LIN {X 0,Y 411.309,Z 303.251,A -85,B 0,C 180,E1 -10615.099,E2 -10615.099} C_VEL
LIN {X 0,Y 411.516,Z 303.227,A -85,B 0,C 180,E1 -10618.042,E2 -10618.042} C_VEL
LIN {X 0,Y 411.646,Z 303.212,A -85,B 0,C 180,E1 -10620,E2 -10620} C_VEL
LIN {X 0,Y 411.47,Z 303.233,A -85,B 0,C 180,E1 -10622.937,E2 -10622.937} C_VEL
LIN {X 0,Y 411.429,Z 303.238,A -85,B 0,C 180,E1 -10626.867,E2 -10626.867} C_VEL
LIN {X 0,Y 411.156,Z 303.275,A -85,B 0,C 180,E1 -10629.842,E2 -10629.842} C_VEL
LIN {X 0,Y 411.049,Z 303.289,A -85,B 0,C 180,E1 -10630.84,E2 -10630.84} C_VEL
LIN {X 0,Y 411.031,Z 303.714,A -85,B 0,C 180,E1 -10631.84,E2 -10631.84} C_VEL
LIN {X 0,Y 410.866,Z 306.355,A -85,B 0,C 180,E1 -10634.867,E2 -10634.867} C_VEL
LIN {X 0,Y 410.709,Z 309.078,A -85,B 0,C 180,E1 -10637.939,E2 -10637.939} C_VEL
LIN {X 0,Y 410.69,Z 311.358,A -85,B 0,C 180,E1 -10640.34,E2 -10640.34} C_VEL
LIN {X 0,Y 414.787,Z 325.038,A -85,B 0,C 180,E1 -10641.071,E2 -10641.071} C_VEL
LIN {X 0,Y 416.146,Z 330.89,A -85,B 0,C 180,E1 -10641.434,E2 -10641.434} C_VEL
LIN {X 0,Y 415.65,Z 342.021,A -85,B 0,C 180,E1 -10642.099,E2 -10642.099} C_VEL
LIN {X 0,Y 414.871,Z 354.086,A -85,B 0,C 180,E1 -10643.037,E2 -10643.037} C_VEL
LIN {X 0,Y 414.058,Z 365.557,A -85,B 0,C 180,E1 -10644.172,E2 -10644.172} C_VEL
LIN {X 0,Y 413.296,Z 375.312,A -85,B 0,C 180,E1 -10645.388,E2 -10645.388} C_VEL
LIN {X 0,Y 412.511,Z 384.696,A -85,B 0,C 180,E1 -10646.839,E2 -10646.839} C_VEL
LIN {X 0,Y 411.876,Z 392.147,A -85,B 0,C 180,E1 -10648.272,E2 -10648.272} C_VEL
LIN {X 0,Y 411.372,Z 398.098,A -85,B 0,C 180,E1 -10649.699,E2 -10649.699} C_VEL
LIN {X 0,Y 410.927,Z 403.134,A -85,B 0,C 180,E1 -10651.224,E2 -10651.224} C_VEL
LIN {X 0,Y 410.575,Z 407.484,A -85,B 0,C 180,E1 -10652.99,E2 -10652.99} C_VEL
LIN {X 0,Y 410.282,Z 410.333,A -85,B 0,C 180,E1 -10654.691,E2 -10654.691} C_VEL
LIN {X 0,Y 410.113,Z 411.91,A -85,B 0,C 180,E1 -10656.348,E2 -10656.348} C_VEL
LIN {X 0,Y 410.08,Z 412.317,A -85,B 0,C 180,E1 -10658.095,E2 -10658.095} C_VEL
LIN {X 0,Y 410.112,Z 411.728,A -85,B 0,C 180,E1 -10659.542,E2 -10659.542} C_VEL
LIN {X 0,Y 410.193,Z 410.148,A -85,B 0,C 180,E1 -10661.073,E2 -10661.073} C_VEL
LIN {X 0,Y 410.43,Z 407.6,A -85,B 0,C 180,E1 -10662.581,E2 -10662.581} C_VEL
LIN {X 0,Y 410.647,Z 404.145,A -85,B 0,C 180,E1 -10664.043,E2 -10664.043} C_VEL
LIN {X 0,Y 410.959,Z 399.707,A -85,B 0,C 180,E1 -10665.479,E2 -10665.479} C_VEL
LIN {X 0,Y 411.253,Z 394.299,A -85,B 0,C 180,E1 -10666.876,E2 -10666.876} C_VEL
LIN {X 0,Y 411.824,Z 386.807,A -85,B 0,C 180,E1 -10668.418,E2 -10668.418} C_VEL
LIN {X 0,Y 412.453,Z 377.956,A -85,B 0,C 180,E1 -10669.879,E2 -10669.879} C_VEL
LIN {X 0,Y 413.129,Z 368.681,A -85,B 0,C 180,E1 -10671.121,E2 -10671.121} C_VEL
LIN {X 0,Y 413.823,Z 358.621,A -85,B 0,C 180,E1 -10672.209,E2 -10672.209} C_VEL
LIN {X 0,Y 414.436,Z 347.453,A -85,B 0,C 180,E1 -10673.186,E2 -10673.186} C_VEL
LIN {X 0,Y 415.151,Z 335.294,A -85,B 0,C 180,E1 -10674.014,E2 -10674.014} C_VEL
LIN {X 0,Y 415.255,Z 328.945,A -85,B 0,C 180,E1 -10674.367,E2 -10674.367} C_VEL
LIN {X 0,Y 412.168,Z 315.956,A -85,B 0,C 180,E1 -10675.058,E2 -10675.058} C_VEL
LIN {X 0,Y 410.372,Z 308.871,A -85,B 0,C 180,E1 -10675.373,E2 -10675.373} C_VEL
LIN {X 0,Y 410.408,Z 305.017,A -85,B 0,C 180,E1 -10679.087,E2 -10679.087} C_VEL
LIN {X 0,Y 410.466,Z 303.359,A -85,B 0,C 180,E1 -10680.835,E2 -10680.835} C_VEL
LIN {X 0,Y 410.797,Z 303.317,A -85,B 0,C 180,E1 -10683.588,E2 -10683.588} C_VEL
LIN {X 0,Y 411.124,Z 303.275,A -85,B 0,C 180,E1 -10686.848,E2 -10686.848} C_VEL
LIN {X 0,Y 411.215,Z 303.26,A -85,B 0,C 180,E1 -10690.051,E2 -10690.051} C_VEL
LIN {X 0,Y 411.264,Z 303.258,A -85,B 0,C 180,E1 -10693.131,E2 -10693.131} C_VEL
LIN {X 0,Y 411.307,Z 303.253,A -85,B 0,C 180,E1 -10696.896,E2 -10696.896} C_VEL
LIN {X 0,Y 411.293,Z 303.252,A -85,B 0,C 180,E1 -10700.161,E2 -10700.161} C_VEL
LIN {X 0,Y 411.424,Z 303.238,A -85,B 0,C 180,E1 -10703.132,E2 -10703.132} C_VEL
LIN {X 0,Y 411.308,Z 303.253,A -85,B 0,C 180,E1 -10705.099,E2 -10705.099} C_VEL
LIN {X 0,Y 411.512,Z 303.225,A -85,B 0,C 180,E1 -10708.043,E2 -10708.043} C_VEL
LIN {X 0,Y 411.642,Z 303.208,A -85,B 0,C 180,E1 -10710,E2 -10710} C_VEL
LIN {X 0,Y 411.467,Z 303.234,A -85,B 0,C 180,E1 -10712.937,E2 -10712.937} C_VEL
LIN {X 0,Y 411.339,Z 303.246,A -85,B 0,C 180,E1 -10715.221,E2 -10715.221} C_VEL
LIN {X 0,Y 410.74,Z 303.323,A -85,B 0,C 180,E1 -10716.039,E2 -10716.039} C_VEL
LIN {X 0,Y 407.884,Z 303.676,A -85,B 0,C 180,E1 -10717.368,E2 -10717.368} C_VEL
LIN {X 0,Y 405.417,Z 303.987,A -85,B 0,C 180,E1 -10718.442,E2 -10718.442} C_VEL
LIN {X 0,Y 404.347,Z 304.117,A -85,B 0,C 180,E1 -10719.272,E2 -10719.272} C_VEL
LIN {X 0,Y 404.257,Z 304.128,A -85,B 0,C 180,E1 -10719.554,E2 -10719.554} C_VEL
LIN {X 0,Y 404.267,Z 304.127,A -85,B 0,C 180,E1 -10723.211,E2 -10723.211} C_VEL
LIN {X 0,Y 404.217,Z 304.134,A -85,B 0,C 180,E1 -10727.007,E2 -10727.007} C_VEL
LIN {X 0,Y 404.165,Z 304.143,A -85,B 0,C 180,E1 -10730.352,E2 -10730.352} C_VEL
LIN {X 0,Y 404.171,Z 304.139,A -85,B 0,C 180,E1 -10733.575,E2 -10733.575} C_VEL
LIN {X 0,Y 404.185,Z 304.139,A -85,B 0,C 180,E1 -10735.767,E2 -10735.767} C_VEL
LIN {X 0,Y 404.196,Z 304.139,A -85,B 0,C 180,E1 -10738,E2 -10738} C_VEL
LIN {X 0,Y 404.14,Z 304.144,A -85,B 0,C 180,E1 -10741.558,E2 -10741.558} C_VEL
LIN {X 0,Y 404.185,Z 304.137,A -85,B 0,C 180,E1 -10745.016,E2 -10745.016} C_VEL
LIN {X 0,Y 404.156,Z 304.141,A -85,B 0,C 180,E1 -10748.757,E2 -10748.757} C_VEL
LIN {X 0,Y 404.125,Z 304.148,A -85,B 0,C 180,E1 -10751.6,E2 -10751.6} C_VEL
LIN {X 0,Y 404.147,Z 304.142,A -85,B 0,C 180,E1 -10754.522,E2 -10754.522} C_VEL
LIN {X 0,Y 404.139,Z 304.144,A -85,B 0,C 180,E1 -10757.296,E2 -10757.296} C_VEL
LIN {X 0,Y 404.171,Z 304.142,A -85,B 0,C 180,E1 -10759.956,E2 -10759.956} C_VEL
LIN {X 0,Y 404.139,Z 304.144,A -85,B 0,C 180,E1 -10763.125,E2 -10763.125} C_VEL
LIN {X 0,Y 404.147,Z 304.142,A -85,B 0,C 180,E1 -10766.188,E2 -10766.188} C_VEL
LIN {X 0,Y 404.149,Z 304.144,A -85,B 0,C 180,E1 -10769.715,E2 -10769.715} C_VEL
LIN {X 0,Y 404.196,Z 304.138,A -85,B 0,C 180,E1 -10773.123,E2 -10773.123} C_VEL
LIN {X 0,Y 404.173,Z 304.142,A -85,B 0,C 180,E1 -10775.334,E2 -10775.334} C_VEL
LIN {X 0,Y 404.142,Z 304.142,A -85,B 0,C 180,E1 -10778.581,E2 -10778.581} C_VEL
LIN {X 0,Y 404.209,Z 304.135,A -85,B 0,C 180,E1 -10781.762,E2 -10781.762} C_VEL
LIN {X 0,Y 404.21,Z 304.136,A -85,B 0,C 180,E1 -10784.882,E2 -10784.882} C_VEL
LIN {X 0,Y 404.261,Z 304.128,A -85,B 0,C 180,E1 -10787.959,E2 -10787.959} C_VEL
LIN {X 0,Y 404.27,Z 304.13,A -85,B 0,C 180,E1 -10790.999,E2 -10790.999} C_VEL
LIN {X 0,Y 404.422,Z 304.107,A -85,B 0,C 180,E1 -10794.015,E2 -10794.015} C_VEL
LIN {X 0,Y 404.483,Z 304.099,A -85,B 0,C 180,E1 -10798.009,E2 -10798.009} C_VEL
LIN {X 0,Y 404.612,Z 304.084,A -85,B 0,C 180,E1 -10800,E2 -10800} C_VEL
LIN {X 0,Y 404.408,Z 304.112,A -85,B 0,C 180,E1 -10802.989,E2 -10802.989} C_VEL
LIN {X 0,Y 404.373,Z 304.116,A -85,B 0,C 180,E1 -10806.988,E2 -10806.988} C_VEL
LIN {X 0,Y 404.261,Z 304.127,A -85,B 0,C 180,E1 -10810.012,E2 -10810.012} C_VEL
LIN {X 0,Y 404.271,Z 304.126,A -85,B 0,C 180,E1 -10813.211,E2 -10813.211} C_VEL
LIN {X 0,Y 404.22,Z 304.133,A -85,B 0,C 180,E1 -10817.007,E2 -10817.007} C_VEL
LIN {X 0,Y 404.168,Z 304.142,A -85,B 0,C 180,E1 -10820.352,E2 -10820.352} C_VEL
LIN {X 0,Y 404.164,Z 304.14,A -85,B 0,C 180,E1 -10823.575,E2 -10823.575} C_VEL
LIN {X 0,Y 404.155,Z 304.142,A -85,B 0,C 180,E1 -10826.88,E2 -10826.88} C_VEL
LIN {X 0,Y 404.148,Z 304.145,A -85,B 0,C 180,E1 -10830.285,E2 -10830.285} C_VEL
LIN {X 0,Y 404.149,Z 304.143,A -85,B 0,C 180,E1 -10833.812,E2 -10833.812} C_VEL
LIN {X 0,Y 404.139,Z 304.142,A -85,B 0,C 180,E1 -10836.875,E2 -10836.875} C_VEL
LIN {X 0,Y 404.151,Z 304.144,A -85,B 0,C 180,E1 -10840.08,E2 -10840.08} C_VEL
LIN {X 0,Y 404.153,Z 304.144,A -85,B 0,C 180,E1 -10843.083,E2 -10843.083} C_VEL
LIN {X 0,Y 404.15,Z 304.142,A -85,B 0,C 180,E1 -10845.926,E2 -10845.926} C_VEL
LIN {X 0,Y 404.171,Z 304.244,A -85,B 0,C 180,E1 -10847.204,E2 -10847.204} C_VEL
LIN {X 0,Y 405.52,Z 311.584,A -85,B 0,C 180,E1 -10850.707,E2 -10850.707} C_VEL
LIN {X 0,Y 406.463,Z 317.496,A -85,B 0,C 180,E1 -10853.378,E2 -10853.378} C_VEL
LIN {X 0,Y 406.168,Z 323.082,A -85,B 0,C 180,E1 -10855.736,E2 -10855.736} C_VEL
LIN {X 0,Y 405.489,Z 330.3,A -85,B 0,C 180,E1 -10858.67,E2 -10858.67} C_VEL
LIN {X 0,Y 404.96,Z 337.41,A -85,B 0,C 180,E1 -10861.493,E2 -10861.493} C_VEL
LIN {X 0,Y 404.381,Z 345.551,A -85,B 0,C 180,E1 -10864.655,E2 -10864.655} C_VEL
LIN {X 0,Y 403.858,Z 354.455,A -85,B 0,C 180,E1 -10868.028,E2 -10868.028} C_VEL
LIN {X 0,Y 403.524,Z 362.939,A -85,B 0,C 180,E1 -10871.203,E2 -10871.203} C_VEL
LIN {X 0,Y 403.416,Z 365.913,A -85,B 0,C 180,E1 -10872.304,E2 -10872.304} C_VEL
LIN {X 0,Y 405.324,Z 379.721,A -85,B 0,C 180,E1 -10872.813,E2 -10872.813} C_VEL
LIN {X 0,Y 406.616,Z 391.696,A -85,B 0,C 180,E1 -10873.425,E2 -10873.425} C_VEL
LIN {X 0,Y 407.147,Z 400.281,A -85,B 0,C 180,E1 -10873.967,E2 -10873.967} C_VEL
LIN {X 0,Y 406.322,Z 411.995,A -85,B 0,C 180,E1 -10874.834,E2 -10874.834} C_VEL
LIN {X 0,Y 405.435,Z 423.753,A -85,B 0,C 180,E1 -10875.955,E2 -10875.955} C_VEL
LIN {X 0,Y 404.729,Z 434.257,A -85,B 0,C 180,E1 -10877.209,E2 -10877.209} C_VEL
LIN {X 0,Y 404.15,Z 442.777,A -85,B 0,C 180,E1 -10878.464,E2 -10878.464} C_VEL
LIN {X 0,Y 403.562,Z 451.09,A -85,B 0,C 180,E1 -10879.971,E2 -10879.971} C_VEL
LIN {X 0,Y 403.285,Z 457.801,A -85,B 0,C 180,E1 -10881.481,E2 -10881.481} C_VEL
LIN {X 0,Y 403.077,Z 463.139,A -85,B 0,C 180,E1 -10882.989,E2 -10882.989} C_VEL
LIN {X 0,Y 403.034,Z 467.281,A -85,B 0,C 180,E1 -10884.496,E2 -10884.496} C_VEL
LIN {X 0,Y 402.964,Z 470.331,A -85,B 0,C 180,E1 -10886,E2 -10886} C_VEL
LIN {X 0,Y 403.09,Z 471.836,A -85,B 0,C 180,E1 -10887.002,E2 -10887.002} C_VEL
LIN {X 0,Y 403.089,Z 472.867,A -85,B 0,C 180,E1 -10888.002,E2 -10888.002} C_VEL
LIN {X 0,Y 403.098,Z 473.495,A -85,B 0,C 180,E1 -10889.001,E2 -10889.001} C_VEL
LIN {X 0,Y 403.069,Z 473.721,A -85,B 0,C 180,E1 -10890,E2 -10890} C_VEL
LIN {X 0,Y 403.097,Z 473.538,A -85,B 0,C 180,E1 -10890.999,E2 -10890.999} C_VEL
LIN {X 0,Y 403.098,Z 471.88,A -85,B 0,C 180,E1 -10892.998,E2 -10892.998} C_VEL
LIN {X 0,Y 402.965,Z 470.435,A -85,B 0,C 180,E1 -10894,E2 -10894} C_VEL
LIN {X 0,Y 402.993,Z 467.431,A -85,B 0,C 180,E1 -10895.504,E2 -10895.504} C_VEL
LIN {X 0,Y 403.076,Z 463.375,A -85,B 0,C 180,E1 -10897.011,E2 -10897.011} C_VEL
LIN {X 0,Y 403.302,Z 457.185,A -85,B 0,C 180,E1 -10898.771,E2 -10898.771} C_VEL
LIN {X 0,Y 403.651,Z 450.416,A -85,B 0,C 180,E1 -10900.28,E2 -10900.28} C_VEL
LIN {X 0,Y 404.289,Z 442.056,A -85,B 0,C 180,E1 -10901.786,E2 -10901.786} C_VEL
LIN {X 0,Y 404.923,Z 433.557,A -85,B 0,C 180,E1 -10903.04,E2 -10903.04} C_VEL
LIN {X 0,Y 405.684,Z 423.173,A -85,B 0,C 180,E1 -10904.292,E2 -10904.292} C_VEL
LIN {X 0,Y 406.678,Z 411.581,A -85,B 0,C 180,E1 -10905.409,E2 -10905.409} C_VEL
LIN {X 0,Y 407.546,Z 400.302,A -85,B 0,C 180,E1 -10906.274,E2 -10906.274} C_VEL
LIN {X 0,Y 406.791,Z 387.739,A -85,B 0,C 180,E1 -10907.08,E2 -10907.08} C_VEL
LIN {X 0,Y 405.258,Z 374.108,A -85,B 0,C 180,E1 -10907.764,E2 -10907.764} C_VEL
LIN {X 0,Y 403.409,Z 363.522,A -85,B 0,C 180,E1 -10908.21,E2 -10908.21} C_VEL
LIN {X 0,Y 403.741,Z 354.769,A -85,B 0,C 180,E1 -10911.442,E2 -10911.442} C_VEL
LIN {X 0,Y 404.156,Z 346.259,A -85,B 0,C 180,E1 -10914.667,E2 -10914.667} C_VEL
LIN {X 0,Y 404.826,Z 336.442,A -85,B 0,C 180,E1 -10918.517,E2 -10918.517} C_VEL
LIN {X 0,Y 405.705,Z 326.904,A -85,B 0,C 180,E1 -10922.481,E2 -10922.481} C_VEL
LIN {X 0,Y 406.508,Z 318.939,A -85,B 0,C 180,E1 -10926.003,E2 -10926.003} C_VEL
LIN {X 0,Y 406.15,Z 315.059,A -85,B 0,C 180,E1 -10927.9,E2 -10927.9} C_VEL
LIN {X 0,Y 405.06,Z 308.803,A -85,B 0,C 180,E1 -10931.248,E2 -10931.248} C_VEL
LIN {X 0,Y 404.152,Z 304.149,A -85,B 0,C 180,E1 -10934.074,E2 -10934.074} C_VEL
LIN {X 0,Y 404.14,Z 304.151,A -85,B 0,C 180,E1 -10937.296,E2 -10937.296} C_VEL
LIN {X 0,Y 404.172,Z 304.144,A -85,B 0,C 180,E1 -10939.955,E2 -10939.955} C_VEL
LIN {X 0,Y 404.14,Z 304.145,A -85,B 0,C 180,E1 -10943.125,E2 -10943.125} C_VEL
LIN {X 0,Y 404.149,Z 304.145,A -85,B 0,C 180,E1 -10946.188,E2 -10946.188} C_VEL
LIN {X 0,Y 404.15,Z 304.144,A -85,B 0,C 180,E1 -10949.715,E2 -10949.715} C_VEL
LIN {X 0,Y 404.2,Z 304.138,A -85,B 0,C 180,E1 -10953.123,E2 -10953.123} C_VEL
LIN {X 0,Y 404.182,Z 304.137,A -85,B 0,C 180,E1 -10955.334,E2 -10955.334} C_VEL
LIN {X 0,Y 404.144,Z 304.145,A -85,B 0,C 180,E1 -10958.581,E2 -10958.581} C_VEL
LIN {X 0,Y 404.213,Z 304.135,A -85,B 0,C 180,E1 -10961.762,E2 -10961.762} C_VEL
LIN {X 0,Y 404.211,Z 304.134,A -85,B 0,C 180,E1 -10964.882,E2 -10964.882} C_VEL
LIN {X 0,Y 404.261,Z 304.131,A -85,B 0,C 180,E1 -10967.958,E2 -10967.958} C_VEL
LIN {X 0,Y 404.271,Z 304.128,A -85,B 0,C 180,E1 -10970.998,E2 -10970.998} C_VEL
LIN {X 0,Y 404.396,Z 304.113,A -85,B 0,C 180,E1 -10974.015,E2 -10974.015} C_VEL
LIN {X 0,Y 404.485,Z 304.103,A -85,B 0,C 180,E1 -10978.008,E2 -10978.008} C_VEL
LIN {X 0,Y 404.615,Z 304.088,A -85,B 0,C 180,E1 -10980,E2 -10980} C_VEL
LIN {X 0,Y 404.427,Z 304.111,A -85,B 0,C 180,E1 -10982.988,E2 -10982.988} C_VEL
LIN {X 0,Y 404.374,Z 304.117,A -85,B 0,C 180,E1 -10986.988,E2 -10986.988} C_VEL
LIN {X 0,Y 404.082,Z 304.156,A -85,B 0,C 180,E1 -10990.016,E2 -10990.016} C_VEL
LIN {X 0,Y 403.981,Z 304.169,A -85,B 0,C 180,E1 -10991.032,E2 -10991.032} C_VEL
LIN {X 0,Y 403.933,Z 305.806,A -85,B 0,C 180,E1 -10993.073,E2 -10993.073} C_VEL
LIN {X 0,Y 403.805,Z 308.477,A -85,B 0,C 180,E1 -10996.169,E2 -10996.169} C_VEL
LIN {X 0,Y 403.644,Z 311.846,A -85,B 0,C 180,E1 -10999.972,E2 -10999.972} C_VEL
LIN {X 0,Y 407.768,Z 325.499,A -85,B 0,C 180,E1 -11000.724,E2 -11000.724} C_VEL
LIN {X 0,Y 409.449,Z 332.857,A -85,B 0,C 180,E1 -11001.194,E2 -11001.194} C_VEL
LIN {X 0,Y 408.798,Z 344.75,A -85,B 0,C 180,E1 -11001.949,E2 -11001.949} C_VEL
LIN {X 0,Y 407.961,Z 356.799,A -85,B 0,C 180,E1 -11002.94,E2 -11002.94} C_VEL
LIN {X 0,Y 407.096,Z 367.899,A -85,B 0,C 180,E1 -11004.111,E2 -11004.111} C_VEL
LIN {X 0,Y 406.301,Z 377.329,A -85,B 0,C 180,E1 -11005.348,E2 -11005.348} C_VEL
LIN {X 0,Y 405.511,Z 386.203,A -85,B 0,C 180,E1 -11006.783,E2 -11006.783} C_VEL
LIN {X 0,Y 404.858,Z 393.389,A -85,B 0,C 180,E1 -11008.232,E2 -11008.232} C_VEL
LIN {X 0,Y 404.244,Z 400.049,A -85,B 0,C 180,E1 -11009.922,E2 -11009.922} C_VEL
LIN {X 0,Y 403.812,Z 404.806,A -85,B 0,C 180,E1 -11011.481,E2 -11011.481} C_VEL
LIN {X 0,Y 403.457,Z 408.806,A -85,B 0,C 180,E1 -11013.265,E2 -11013.265} C_VEL
LIN {X 0,Y 403.152,Z 411.47,A -85,B 0,C 180,E1 -11015.119,E2 -11015.119} C_VEL
LIN {X 0,Y 403.038,Z 412.625,A -85,B 0,C 180,E1 -11016.666,E2 -11016.666} C_VEL
LIN {X 0,Y 403.001,Z 412.81,A -85,B 0,C 180,E1 -11018.301,E2 -11018.301} C_VEL
LIN {X 0,Y 403.059,Z 411.724,A -85,B 0,C 180,E1 -11020.177,E2 -11020.177} C_VEL
LIN {X 0,Y 403.264,Z 409.029,A -85,B 0,C 180,E1 -11022.142,E2 -11022.142} C_VEL
LIN {X 0,Y 403.522,Z 406.175,A -85,B 0,C 180,E1 -11023.518,E2 -11023.518} C_VEL
LIN {X 0,Y 403.771,Z 402.298,A -85,B 0,C 180,E1 -11024.941,E2 -11024.941} C_VEL
LIN {X 0,Y 404.115,Z 396.265,A -85,B 0,C 180,E1 -11026.641,E2 -11026.641} C_VEL
LIN {X 0,Y 404.707,Z 388.687,A -85,B 0,C 180,E1 -11028.307,E2 -11028.307} C_VEL
LIN {X 0,Y 405.314,Z 380.596,A -85,B 0,C 180,E1 -11029.724,E2 -11029.724} C_VEL
LIN {X 0,Y 406.092,Z 370.467,A -85,B 0,C 180,E1 -11031.15,E2 -11031.15} C_VEL
LIN {X 0,Y 406.787,Z 360.994,A -85,B 0,C 180,E1 -11032.231,E2 -11032.231} C_VEL
LIN {X 0,Y 407.493,Z 349.174,A -85,B 0,C 180,E1 -11033.314,E2 -11033.314} C_VEL
LIN {X 0,Y 408.246,Z 337.049,A -85,B 0,C 180,E1 -11034.174,E2 -11034.174} C_VEL
LIN {X 0,Y 408.438,Z 330.329,A -85,B 0,C 180,E1 -11034.567,E2 -11034.567} C_VEL
LIN {X 0,Y 405.471,Z 317.829,A -85,B 0,C 180,E1 -11035.262,E2 -11035.262} C_VEL
LIN {X 0,Y 403.314,Z 309.34,A -85,B 0,C 180,E1 -11035.656,E2 -11035.656} C_VEL
LIN {X 0,Y 403.318,Z 306.271,A -85,B 0,C 180,E1 -11038.633,E2 -11038.633} C_VEL
LIN {X 0,Y 403.42,Z 304.237,A -85,B 0,C 180,E1 -11040.804,E2 -11040.804} C_VEL
LIN {X 0,Y 403.718,Z 304.199,A -85,B 0,C 180,E1 -11043.088,E2 -11043.088} C_VEL
LIN {X 0,Y 403.948,Z 304.171,A -85,B 0,C 180,E1 -11045.319,E2 -11045.319} C_VEL
LIN {X 0,Y 404.145,Z 304.144,A -85,B 0,C 180,E1 -11047.506,E2 -11047.506} C_VEL
LIN {X 0,Y 404.163,Z 304.141,A -85,B 0,C 180,E1 -11050.707,E2 -11050.707} C_VEL
LIN {X 0,Y 404.222,Z 304.132,A -85,B 0,C 180,E1 -11053.848,E2 -11053.848} C_VEL
LIN {X 0,Y 404.284,Z 304.128,A -85,B 0,C 180,E1 -11056.939,E2 -11056.939} C_VEL
LIN {X 0,Y 404.259,Z 304.128,A -85,B 0,C 180,E1 -11059.988,E2 -11059.988} C_VEL
LIN {X 0,Y 404.37,Z 304.117,A -85,B 0,C 180,E1 -11063.012,E2 -11063.012} C_VEL
LIN {X 0,Y 404.278,Z 304.129,A -85,B 0,C 180,E1 -11065.013,E2 -11065.013} C_VEL
LIN {X 0,Y 404.481,Z 304.101,A -85,B 0,C 180,E1 -11068.008,E2 -11068.008} C_VEL
LIN {X 0,Y 404.611,Z 304.084,A -85,B 0,C 180,E1 -11070,E2 -11070} C_VEL
LIN {X 0,Y 404.424,Z 304.11,A -85,B 0,C 180,E1 -11072.988,E2 -11072.988} C_VEL
LIN {X 0,Y 404.37,Z 304.116,A -85,B 0,C 180,E1 -11076.988,E2 -11076.988} C_VEL
LIN {X 0,Y 404.257,Z 304.128,A -85,B 0,C 180,E1 -11079.554,E2 -11079.554} C_VEL
LIN {X 0,Y 403.584,Z 304.215,A -85,B 0,C 180,E1 -11080.385,E2 -11080.385} C_VEL
LIN {X 0,Y 400.732,Z 304.567,A -85,B 0,C 180,E1 -11081.737,E2 -11081.737} C_VEL
LIN {X 0,Y 398.316,Z 304.87,A -85,B 0,C 180,E1 -11082.829,E2 -11082.829} C_VEL
LIN {X 0,Y 397.271,Z 304.998,A -85,B 0,C 180,E1 -11083.674,E2 -11083.674} C_VEL
LIN {X 0,Y 397.181,Z 305.009,A -85,B 0,C 180,E1 -11083.96,E2 -11083.96} C_VEL
LIN {X 0,Y 397.175,Z 305.01,A -85,B 0,C 180,E1 -11087.507,E2 -11087.507} C_VEL
LIN {X 0,Y 397.104,Z 305.021,A -85,B 0,C 180,E1 -11090.73,E2 -11090.73} C_VEL
LIN {X 0,Y 397.135,Z 305.018,A -85,B 0,C 180,E1 -11094.018,E2 -11094.018} C_VEL
LIN {X 0,Y 397.196,Z 305.007,A -85,B 0,C 180,E1 -11097.39,E2 -11097.39} C_VEL
LIN {X 0,Y 397.079,Z 305.022,A -85,B 0,C 180,E1 -11100.883,E2 -11100.883} C_VEL
LIN {X 0,Y 397.126,Z 305.018,A -85,B 0,C 180,E1 -11104.494,E2 -11104.494} C_VEL
LIN {X 0,Y 397.104,Z 305.022,A -85,B 0,C 180,E1 -11108.275,E2 -11108.275} C_VEL
LIN {X 0,Y 397.09,Z 305.02,A -85,B 0,C 180,E1 -11110.909,E2 -11110.909} C_VEL
LIN {X 0,Y 397.103,Z 305.022,A -85,B 0,C 180,E1 -11113.649,E2 -11113.649} C_VEL
LIN {X 0,Y 397.104,Z 305.019,A -85,B 0,C 180,E1 -11116.521,E2 -11116.521} C_VEL
LIN {X 0,Y 397.117,Z 305.018,A -85,B 0,C 180,E1 -11120.423,E2 -11120.423} C_VEL
LIN {X 0,Y 397.11,Z 305.019,A -85,B 0,C 180,E1 -11124.266,E2 -11124.266} C_VEL
LIN {X 0,Y 397.117,Z 305.017,A -85,B 0,C 180,E1 -11126.727,E2 -11126.727} C_VEL
LIN {X 0,Y 397.127,Z 305.016,A -85,B 0,C 180,E1 -11130.296,E2 -11130.296} C_VEL
LIN {X 0,Y 397.197,Z 305.007,A -85,B 0,C 180,E1 -11132.61,E2 -11132.61} C_VEL
LIN {X 0,Y 397.129,Z 305.017,A -85,B 0,C 180,E1 -11135.982,E2 -11135.982} C_VEL
LIN {X 0,Y 397.142,Z 305.017,A -85,B 0,C 180,E1 -11139.705,E2 -11139.705} C_VEL
LIN {X 0,Y 397.186,Z 305.011,A -85,B 0,C 180,E1 -11142.845,E2 -11142.845} C_VEL
LIN {X 0,Y 397.233,Z 305.004,A -85,B 0,C 180,E1 -11146.703,E2 -11146.703} C_VEL
LIN {X 0,Y 397.221,Z 305.004,A -85,B 0,C 180,E1 -11149.809,E2 -11149.809} C_VEL
LIN {X 0,Y 397.342,Z 304.992,A -85,B 0,C 180,E1 -11152.888,E2 -11152.888} C_VEL
LIN {X 0,Y 397.256,Z 305.004,A -85,B 0,C 180,E1 -11154.925,E2 -11154.925} C_VEL
LIN {X 0,Y 397.452,Z 304.975,A -85,B 0,C 180,E1 -11157.973,E2 -11157.973} C_VEL
LIN {X 0,Y 397.581,Z 304.96,A -85,B 0,C 180,E1 -11160,E2 -11160} C_VEL
LIN {X 0,Y 397.342,Z 304.992,A -85,B 0,C 180,E1 -11163.042,E2 -11163.042} C_VEL
LIN {X 0,Y 397.348,Z 304.988,A -85,B 0,C 180,E1 -11166.092,E2 -11166.092} C_VEL
LIN {X 0,Y 397.24,Z 305.003,A -85,B 0,C 180,E1 -11169.162,E2 -11169.162} C_VEL
LIN {X 0,Y 397.224,Z 305.007,A -85,B 0,C 180,E1 -11172.258,E2 -11172.258} C_VEL
LIN {X 0,Y 397.183,Z 305.009,A -85,B 0,C 180,E1 -11175.392,E2 -11175.392} C_VEL
LIN {X 0,Y 397.162,Z 305.015,A -85,B 0,C 180,E1 -11178.574,E2 -11178.574} C_VEL
LIN {X 0,Y 397.1,Z 305.019,A -85,B 0,C 180,E1 -11181.818,E2 -11181.818} C_VEL
LIN {X 0,Y 397.127,Z 305.015,A -85,B 0,C 180,E1 -11185.134,E2 -11185.134} C_VEL
LIN {X 0,Y 397.103,Z 305.022,A -85,B 0,C 180,E1 -11188.545,E2 -11188.545} C_VEL
LIN {X 0,Y 397.082,Z 305.025,A -85,B 0,C 180,E1 -11192.071,E2 -11192.071} C_VEL
LIN {X 0,Y 397.123,Z 305.018,A -85,B 0,C 180,E1 -11195.503,E2 -11195.503} C_VEL
LIN {X 0,Y 397.128,Z 305.016,A -85,B 0,C 180,E1 -11198.86,E2 -11198.86} C_VEL
LIN {X 0,Y 397.068,Z 305.026,A -85,B 0,C 180,E1 -11202.268,E2 -11202.268} C_VEL
LIN {X 0,Y 397.09,Z 305.021,A -85,B 0,C 180,E1 -11205.069,E2 -11205.069} C_VEL
LIN {X 0,Y 397.135,Z 305.125,A -85,B 0,C 180,E1 -11206.915,E2 -11206.915} C_VEL
LIN {X 0,Y 398.297,Z 311.423,A -85,B 0,C 180,E1 -11209.997,E2 -11209.997} C_VEL
LIN {X 0,Y 399.203,Z 316.543,A -85,B 0,C 180,E1 -11212.395,E2 -11212.395} C_VEL
LIN {X 0,Y 399.474,Z 320.201,A -85,B 0,C 180,E1 -11214.027,E2 -11214.027} C_VEL
LIN {X 0,Y 398.797,Z 328.225,A -85,B 0,C 180,E1 -11217.401,E2 -11217.401} C_VEL
LIN {X 0,Y 398.011,Z 336.929,A -85,B 0,C 180,E1 -11220.949,E2 -11220.949} C_VEL
LIN {X 0,Y 397.341,Z 345.686,A -85,B 0,C 180,E1 -11224.432,E2 -11224.432} C_VEL
LIN {X 0,Y 396.836,Z 353.898,A -85,B 0,C 180,E1 -11227.619,E2 -11227.619} C_VEL
LIN {X 0,Y 396.402,Z 363.804,A -85,B 0,C 180,E1 -11231.39,E2 -11231.39} C_VEL
LIN {X 0,Y 396.335,Z 365.45,A -85,B 0,C 180,E1 -11232.014,E2 -11232.014} C_VEL
LIN {X 0,Y 398.363,Z 379.828,A -85,B 0,C 180,E1 -11232.565,E2 -11232.565} C_VEL
LIN {X 0,Y 399.717,Z 393.011,A -85,B 0,C 180,E1 -11233.275,E2 -11233.275} C_VEL
LIN {X 0,Y 400.163,Z 401.143,A -85,B 0,C 180,E1 -11233.811,E2 -11233.811} C_VEL
LIN {X 0,Y 399.315,Z 412.488,A -85,B 0,C 180,E1 -11234.692,E2 -11234.692} C_VEL
LIN {X 0,Y 398.386,Z 424.219,A -85,B 0,C 180,E1 -11235.849,E2 -11235.849} C_VEL
LIN {X 0,Y 397.779,Z 433.458,A -85,B 0,C 180,E1 -11236.981,E2 -11236.981} C_VEL
LIN {X 0,Y 397.147,Z 442.037,A -85,B 0,C 180,E1 -11238.258,E2 -11238.258} C_VEL
LIN {X 0,Y 396.499,Z 450.384,A -85,B 0,C 180,E1 -11239.79,E2 -11239.79} C_VEL
LIN {X 0,Y 396.205,Z 457.127,A -85,B 0,C 180,E1 -11241.328,E2 -11241.328} C_VEL
LIN {X 0,Y 396.005,Z 462.496,A -85,B 0,C 180,E1 -11242.864,E2 -11242.864} C_VEL
LIN {X 0,Y 395.949,Z 466.665,A -85,B 0,C 180,E1 -11244.398,E2 -11244.398} C_VEL
LIN {X 0,Y 395.882,Z 469.739,A -85,B 0,C 180,E1 -11245.928,E2 -11245.928} C_VEL
LIN {X 0,Y 396.002,Z 471.26,A -85,B 0,C 180,E1 -11246.948,E2 -11246.948} C_VEL
LIN {X 0,Y 396.015,Z 472.305,A -85,B 0,C 180,E1 -11247.966,E2 -11247.966} C_VEL
LIN {X 0,Y 396.046,Z 472.944,A -85,B 0,C 180,E1 -11248.983,E2 -11248.983} C_VEL
LIN {X 0,Y 396.016,Z 473.178,A -85,B 0,C 180,E1 -11250,E2 -11250} C_VEL
LIN {X 0,Y 396.028,Z 473.007,A -85,B 0,C 180,E1 -11251.017,E2 -11251.017} C_VEL
LIN {X 0,Y 395.998,Z 472.387,A -85,B 0,C 180,E1 -11252.034,E2 -11252.034} C_VEL
LIN {X 0,Y 396.01,Z 471.366,A -85,B 0,C 180,E1 -11253.052,E2 -11253.052} C_VEL
LIN {X 0,Y 395.883,Z 469.925,A -85,B 0,C 180,E1 -11254.072,E2 -11254.072} C_VEL
LIN {X 0,Y 395.894,Z 466.933,A -85,B 0,C 180,E1 -11255.603,E2 -11255.603} C_VEL
LIN {X 0,Y 396.004,Z 462.892,A -85,B 0,C 180,E1 -11257.136,E2 -11257.136} C_VEL
LIN {X 0,Y 396.22,Z 456.723,A -85,B 0,C 180,E1 -11258.929,E2 -11258.929} C_VEL
LIN {X 0,Y 396.601,Z 449.97,A -85,B 0,C 180,E1 -11260.465,E2 -11260.465} C_VEL
LIN {X 0,Y 397.314,Z 441.644,A -85,B 0,C 180,E1 -11261.996,E2 -11261.996} C_VEL
LIN {X 0,Y 398.098,Z 432.082,A -85,B 0,C 180,E1 -11263.425,E2 -11263.425} C_VEL
LIN {X 0,Y 398.861,Z 421.734,A -85,B 0,C 180,E1 -11264.672,E2 -11264.672} C_VEL
LIN {X 0,Y 399.964,Z 409.986,A -85,B 0,C 180,E1 -11265.805,E2 -11265.805} C_VEL
LIN {X 0,Y 400.669,Z 400.225,A -85,B 0,C 180,E1 -11266.561,E2 -11266.561} C_VEL
LIN {X 0,Y 399.967,Z 387.905,A -85,B 0,C 180,E1 -11267.381,E2 -11267.381} C_VEL
LIN {X 0,Y 398.35,Z 374.086,A -85,B 0,C 180,E1 -11268.103,E2 -11268.103} C_VEL
LIN {X 0,Y 396.351,Z 362.938,A -85,B 0,C 180,E1 -11268.583,E2 -11268.583} C_VEL
LIN {X 0,Y 396.715,Z 354.333,A -85,B 0,C 180,E1 -11271.841,E2 -11271.841} C_VEL
LIN {X 0,Y 397.224,Z 344.856,A -85,B 0,C 180,E1 -11275.533,E2 -11275.533} C_VEL
LIN {X 0,Y 397.872,Z 336.152,A -85,B 0,C 180,E1 -11279.063,E2 -11279.063} C_VEL
LIN {X 0,Y 398.723,Z 327.827,A -85,B 0,C 180,E1 -11282.592,E2 -11282.592} C_VEL
LIN {X 0,Y 399.502,Z 320.325,A -85,B 0,C 180,E1 -11285.979,E2 -11285.979} C_VEL
LIN {X 0,Y 399.165,Z 316.204,A -85,B 0,C 180,E1 -11288.042,E2 -11288.042} C_VEL
LIN {X 0,Y 398.11,Z 310.055,A -85,B 0,C 180,E1 -11291.427,E2 -11291.427} C_VEL
LIN {X 0,Y 397.113,Z 305.025,A -85,B 0,C 180,E1 -11294.598,E2 -11294.598} C_VEL
LIN {X 0,Y 397.07,Z 305.032,A -85,B 0,C 180,E1 -11298.021,E2 -11298.021} C_VEL
LIN {X 0,Y 397.135,Z 305.021,A -85,B 0,C 180,E1 -11301.138,E2 -11301.138} C_VEL
LIN {X 0,Y 397.123,Z 305.02,A -85,B 0,C 180,E1 -11304.497,E2 -11304.497} C_VEL
LIN {X 0,Y 397.083,Z 305.025,A -85,B 0,C 180,E1 -11307.929,E2 -11307.929} C_VEL
LIN {X 0,Y 397.127,Z 305.019,A -85,B 0,C 180,E1 -11311.457,E2 -11311.457} C_VEL
LIN {X 0,Y 397.157,Z 305.015,A -85,B 0,C 180,E1 -11314.488,E2 -11314.488} C_VEL
LIN {X 0,Y 397.114,Z 305.02,A -85,B 0,C 180,E1 -11317.086,E2 -11317.086} C_VEL
LIN {X 0,Y 397.152,Z 305.014,A -85,B 0,C 180,E1 -11320.353,E2 -11320.353} C_VEL
LIN {X 0,Y 397.171,Z 305.013,A -85,B 0,C 180,E1 -11323.553,E2 -11323.553} C_VEL
LIN {X 0,Y 397.233,Z 305.003,A -85,B 0,C 180,E1 -11326.703,E2 -11326.703} C_VEL
LIN {X 0,Y 397.222,Z 305.007,A -85,B 0,C 180,E1 -11329.809,E2 -11329.809} C_VEL
LIN {X 0,Y 397.322,Z 304.994,A -85,B 0,C 180,E1 -11332.887,E2 -11332.887} C_VEL
LIN {X 0,Y 397.25,Z 305.003,A -85,B 0,C 180,E1 -11334.925,E2 -11334.925} C_VEL
LIN {X 0,Y 397.454,Z 304.979,A -85,B 0,C 180,E1 -11337.973,E2 -11337.973} C_VEL
LIN {X 0,Y 397.584,Z 304.963,A -85,B 0,C 180,E1 -11340,E2 -11340} C_VEL
LIN {X 0,Y 397.386,Z 304.988,A -85,B 0,C 180,E1 -11343.041,E2 -11343.041} C_VEL
LIN {X 0,Y 397.323,Z 304.996,A -85,B 0,C 180,E1 -11347.112,E2 -11347.112} C_VEL
LIN {X 0,Y 397.024,Z 305.036,A -85,B 0,C 180,E1 -11350.196,E2 -11350.196} C_VEL
LIN {X 0,Y 396.942,Z 305.292,A -85,B 0,C 180,E1 -11351.231,E2 -11351.231} C_VEL
LIN {X 0,Y 396.886,Z 307.027,A -85,B 0,C 180,E1 -11353.309,E2 -11353.309} C_VEL
LIN {X 0,Y 396.76,Z 309.724,A -85,B 0,C 180,E1 -11356.464,E2 -11356.464} C_VEL
LIN {X 0,Y 396.632,Z 312.45,A -85,B 0,C 180,E1 -11359.573,E2 -11359.573} C_VEL
LIN {X 0,Y 401.038,Z 326.782,A -85,B 0,C 180,E1 -11360.417,E2 -11360.417} C_VEL
LIN {X 0,Y 402.484,Z 332.651,A -85,B 0,C 180,E1 -11360.808,E2 -11360.808} C_VEL
LIN {X 0,Y 402.513,Z 338.457,A -85,B 0,C 180,E1 -11361.166,E2 -11361.166} C_VEL
LIN {X 0,Y 401.755,Z 350.099,A -85,B 0,C 180,E1 -11362.005,E2 -11362.005} C_VEL
LIN {X 0,Y 400.849,Z 361.926,A -85,B 0,C 180,E1 -11363.097,E2 -11363.097} C_VEL
LIN {X 0,Y 399.935,Z 372.234,A -85,B 0,C 180,E1 -11364.301,E2 -11364.301} C_VEL
LIN {X 0,Y 399.139,Z 380.945,A -85,B 0,C 180,E1 -11365.556,E2 -11365.556} C_VEL
LIN {X 0,Y 398.391,Z 389.202,A -85,B 0,C 180,E1 -11367.017,E2 -11367.017} C_VEL
LIN {X 0,Y 397.7,Z 395.985,A -85,B 0,C 180,E1 -11368.498,E2 -11368.498} C_VEL
LIN {X 0,Y 397.204,Z 401.104,A -85,B 0,C 180,E1 -11369.888,E2 -11369.888} C_VEL
LIN {X 0,Y 396.701,Z 406.388,A -85,B 0,C 180,E1 -11371.747,E2 -11371.747} C_VEL
LIN {X 0,Y 396.347,Z 410.028,A -85,B 0,C 180,E1 -11373.549,E2 -11373.549} C_VEL
LIN {X 0,Y 396.058,Z 412.278,A -85,B 0,C 180,E1 -11375.287,E2 -11375.287} C_VEL
LIN {X 0,Y 395.938,Z 413.362,A -85,B 0,C 180,E1 -11377.122,E2 -11377.122} C_VEL
LIN {X 0,Y 395.921,Z 413.271,A -85,B 0,C 180,E1 -11378.643,E2 -11378.643} C_VEL
LIN {X 0,Y 395.999,Z 412.197,A -85,B 0,C 180,E1 -11380.257,E2 -11380.257} C_VEL
LIN {X 0,Y 396.13,Z 410.173,A -85,B 0,C 180,E1 -11381.827,E2 -11381.827} C_VEL
LIN {X 0,Y 396.483,Z 406.329,A -85,B 0,C 180,E1 -11383.734,E2 -11383.734} C_VEL
LIN {X 0,Y 396.753,Z 402.544,A -85,B 0,C 180,E1 -11385.117,E2 -11385.117} C_VEL
LIN {X 0,Y 397.14,Z 396.451,A -85,B 0,C 180,E1 -11386.842,E2 -11386.842} C_VEL
LIN {X 0,Y 397.619,Z 390.115,A -85,B 0,C 180,E1 -11388.267,E2 -11388.267} C_VEL
LIN {X 0,Y 398.253,Z 382.358,A -85,B 0,C 180,E1 -11389.691,E2 -11389.691} C_VEL
LIN {X 0,Y 398.986,Z 373.072,A -85,B 0,C 180,E1 -11391.072,E2 -11391.072} C_VEL
LIN {X 0,Y 399.788,Z 362.965,A -85,B 0,C 180,E1 -11392.285,E2 -11392.285} C_VEL
LIN {X 0,Y 400.492,Z 351.81,A -85,B 0,C 180,E1 -11393.37,E2 -11393.37} C_VEL
LIN {X 0,Y 401.281,Z 339.849,A -85,B 0,C 180,E1 -11394.272,E2 -11394.272} C_VEL
LIN {X 0,Y 401.618,Z 332.428,A -85,B 0,C 180,E1 -11394.727,E2 -11394.727} C_VEL
LIN {X 0,Y 399.03,Z 320.605,A -85,B 0,C 180,E1 -11395.426,E2 -11395.426} C_VEL
LIN {X 0,Y 396.262,Z 309.821,A -85,B 0,C 180,E1 -11395.941,E2 -11395.941} C_VEL
LIN {X 0,Y 396.259,Z 306.624,A -85,B 0,C 180,E1 -11399.046,E2 -11399.046} C_VEL
LIN {X 0,Y 396.3,Z 305.31,A -85,B 0,C 180,E1 -11400.339,E2 -11400.339} C_VEL
LIN {X 0,Y 396.62,Z 305.082,A -85,B 0,C 180,E1 -11402.567,E2 -11402.567} C_VEL
LIN {X 0,Y 396.875,Z 305.05,A -85,B 0,C 180,E1 -11404.849,E2 -11404.849} C_VEL
LIN {X 0,Y 397.054,Z 305.029,A -85,B 0,C 180,E1 -11407.082,E2 -11407.082} C_VEL
LIN {X 0,Y 397.147,Z 305.013,A -85,B 0,C 180,E1 -11410.353,E2 -11410.353} C_VEL
LIN {X 0,Y 397.167,Z 305.012,A -85,B 0,C 180,E1 -11413.553,E2 -11413.553} C_VEL
LIN {X 0,Y 397.23,Z 305.006,A -85,B 0,C 180,E1 -11416.703,E2 -11416.703} C_VEL
LIN {X 0,Y 397.218,Z 305.005,A -85,B 0,C 180,E1 -11419.809,E2 -11419.809} C_VEL
LIN {X 0,Y 397.319,Z 304.996,A -85,B 0,C 180,E1 -11422.887,E2 -11422.887} C_VEL
LIN {X 0,Y 397.248,Z 305.004,A -85,B 0,C 180,E1 -11424.925,E2 -11424.925} C_VEL
LIN {X 0,Y 397.45,Z 304.976,A -85,B 0,C 180,E1 -11427.973,E2 -11427.973} C_VEL
LIN {X 0,Y 397.58,Z 304.959,A -85,B 0,C 180,E1 -11430,E2 -11430} C_VEL
LIN {X 0,Y 397.382,Z 304.987,A -85,B 0,C 180,E1 -11433.041,E2 -11433.041} C_VEL
LIN {X 0,Y 397.318,Z 304.993,A -85,B 0,C 180,E1 -11437.113,E2 -11437.113} C_VEL
LIN {X 0,Y 397.218,Z 305.008,A -85,B 0,C 180,E1 -11440.191,E2 -11440.191} C_VEL
LIN {X 0,Y 397.228,Z 305.004,A -85,B 0,C 180,E1 -11443.321,E2 -11443.321} C_VEL
LIN {X 0,Y 397.181,Z 305.009,A -85,B 0,C 180,E1 -11443.96,E2 -11443.96} C_VEL
LIN {X 0,Y 396.499,Z 305.098,A -85,B 0,C 180,E1 -11444.807,E2 -11444.807} C_VEL
LIN {X 0,Y 393.635,Z 305.454,A -85,B 0,C 180,E1 -11446.183,E2 -11446.183} C_VEL
LIN {X 0,Y 391.219,Z 305.752,A -85,B 0,C 180,E1 -11447.295,E2 -11447.295} C_VEL
LIN {X 0,Y 390.183,Z 305.884,A -85,B 0,C 180,E1 -11448.155,E2 -11448.155} C_VEL
LIN {X 0,Y 390.098,Z 305.89,A -85,B 0,C 180,E1 -11448.446,E2 -11448.446} C_VEL
LIN {X 0,Y 390.057,Z 305.897,A -85,B 0,C 180,E1 -11451.122,E2 -11451.122} C_VEL
LIN {X 0,Y 390.082,Z 305.896,A -85,B 0,C 180,E1 -11454.481,E2 -11454.481} C_VEL
LIN {X 0,Y 390.118,Z 305.892,A -85,B 0,C 180,E1 -11457.93,E2 -11457.93} C_VEL
LIN {X 0,Y 390.025,Z 305.901,A -85,B 0,C 180,E1 -11461.505,E2 -11461.505} C_VEL
LIN {X 0,Y 390.086,Z 305.893,A -85,B 0,C 180,E1 -11465.207,E2 -11465.207} C_VEL
LIN {X 0,Y 390.071,Z 305.895,A -85,B 0,C 180,E1 -11469.218,E2 -11469.218} C_VEL
LIN {X 0,Y 390.044,Z 305.9,A -85,B 0,C 180,E1 -11472.374,E2 -11472.374} C_VEL
LIN {X 0,Y 390.046,Z 305.9,A -85,B 0,C 180,E1 -11475.355,E2 -11475.355} C_VEL
LIN {X 0,Y 390.034,Z 305.901,A -85,B 0,C 180,E1 -11478.187,E2 -11478.187} C_VEL
LIN {X 0,Y 390.094,Z 305.892,A -85,B 0,C 180,E1 -11480.908,E2 -11480.908} C_VEL
LIN {X 0,Y 390.087,Z 305.893,A -85,B 0,C 180,E1 -11484.793,E2 -11484.793} C_VEL
LIN {X 0,Y 390.026,Z 305.9,A -85,B 0,C 180,E1 -11488.496,E2 -11488.496} C_VEL
LIN {X 0,Y 390.12,Z 305.89,A -85,B 0,C 180,E1 -11492.07,E2 -11492.07} C_VEL
LIN {X 0,Y 390.078,Z 305.897,A -85,B 0,C 180,E1 -11495.519,E2 -11495.519} C_VEL
LIN {X 0,Y 390.091,Z 305.896,A -85,B 0,C 180,E1 -11499.53,E2 -11499.53} C_VEL
LIN {X 0,Y 390.142,Z 305.889,A -85,B 0,C 180,E1 -11503.248,E2 -11503.248} C_VEL
LIN {X 0,Y 390.198,Z 305.879,A -85,B 0,C 180,E1 -11506.562,E2 -11506.562} C_VEL
LIN {X 0,Y 390.172,Z 305.883,A -85,B 0,C 180,E1 -11509.623,E2 -11509.623} C_VEL
LIN {X 0,Y 390.289,Z 305.87,A -85,B 0,C 180,E1 -11512.759,E2 -11512.759} C_VEL
LIN {X 0,Y 390.228,Z 305.879,A -85,B 0,C 180,E1 -11514.834,E2 -11514.834} C_VEL
LIN {X 0,Y 390.421,Z 305.85,A -85,B 0,C 180,E1 -11517.937,E2 -11517.937} C_VEL
LIN {X 0,Y 390.551,Z 305.835,A -85,B 0,C 180,E1 -11520,E2 -11520} C_VEL
LIN {X 0,Y 390.278,Z 305.872,A -85,B 0,C 180,E1 -11523.097,E2 -11523.097} C_VEL
LIN {X 0,Y 390.303,Z 305.866,A -85,B 0,C 180,E1 -11526.202,E2 -11526.202} C_VEL
LIN {X 0,Y 390.198,Z 305.879,A -85,B 0,C 180,E1 -11529.329,E2 -11529.329} C_VEL
LIN {X 0,Y 390.175,Z 305.885,A -85,B 0,C 180,E1 -11532.483,E2 -11532.483} C_VEL
LIN {X 0,Y 390.143,Z 305.886,A -85,B 0,C 180,E1 -11535.677,E2 -11535.677} C_VEL
LIN {X 0,Y 390.107,Z 305.893,A -85,B 0,C 180,E1 -11538.922,E2 -11538.922} C_VEL
LIN {X 0,Y 390.042,Z 305.902,A -85,B 0,C 180,E1 -11542.234,E2 -11542.234} C_VEL
LIN {X 0,Y 390.088,Z 305.893,A -85,B 0,C 180,E1 -11545.733,E2 -11545.733} C_VEL
LIN {X 0,Y 390.047,Z 305.897,A -85,B 0,C 180,E1 -11549.111,E2 -11549.111} C_VEL
LIN {X 0,Y 390.047,Z 305.899,A -85,B 0,C 180,E1 -11552.721,E2 -11552.721} C_VEL
LIN {X 0,Y 390.059,Z 305.899,A -85,B 0,C 180,E1 -11555.825,E2 -11555.825} C_VEL
LIN {X 0,Y 390.069,Z 305.895,A -85,B 0,C 180,E1 -11559.218,E2 -11559.218} C_VEL
LIN {X 0,Y 390.042,Z 305.901,A -85,B 0,C 180,E1 -11562.373,E2 -11562.373} C_VEL
LIN {X 0,Y 390.047,Z 305.898,A -85,B 0,C 180,E1 -11565.354,E2 -11565.354} C_VEL
LIN {X 0,Y 390.111,Z 306.094,A -85,B 0,C 180,E1 -11566.672,E2 -11566.672} C_VEL
LIN {X 0,Y 391.226,Z 312.167,A -85,B 0,C 180,E1 -11569.706,E2 -11569.706} C_VEL
LIN {X 0,Y 392.243,Z 317.963,A -85,B 0,C 180,E1 -11572.468,E2 -11572.468} C_VEL
LIN {X 0,Y 392.391,Z 322.25,A -85,B 0,C 180,E1 -11574.401,E2 -11574.401} C_VEL
LIN {X 0,Y 391.73,Z 329.45,A -85,B 0,C 180,E1 -11577.482,E2 -11577.482} C_VEL
LIN {X 0,Y 390.957,Z 337.829,A -85,B 0,C 180,E1 -11580.963,E2 -11580.963} C_VEL
LIN {X 0,Y 390.272,Z 346.296,A -85,B 0,C 180,E1 -11584.393,E2 -11584.393} C_VEL
LIN {X 0,Y 389.746,Z 354.773,A -85,B 0,C 180,E1 -11587.748,E2 -11587.748} C_VEL
LIN {X 0,Y 389.305,Z 364.599,A -85,B 0,C 180,E1 -11591.583,E2 -11591.583} C_VEL
LIN {X 0,Y 389.294,Z 364.951,A -85,B 0,C 180,E1 -11591.719,E2 -11591.719} C_VEL
LIN {X 0,Y 391.242,Z 379.03,A -85,B 0,C 180,E1 -11592.265,E2 -11592.265} C_VEL
LIN {X 0,Y 392.703,Z 392.536,A -85,B 0,C 180,E1 -11593.01,E2 -11593.01} C_VEL
LIN {X 0,Y 393.189,Z 401.889,A -85,B 0,C 180,E1 -11593.649,E2 -11593.649} C_VEL
LIN {X 0,Y 392.227,Z 414.395,A -85,B 0,C 180,E1 -11594.675,E2 -11594.675} C_VEL
LIN {X 0,Y 391.309,Z 425.236,A -85,B 0,C 180,E1 -11595.806,E2 -11595.806} C_VEL
LIN {X 0,Y 390.646,Z 434.5,A -85,B 0,C 180,E1 -11597.004,E2 -11597.004} C_VEL
LIN {X 0,Y 389.914,Z 444.292,A -85,B 0,C 180,E1 -11598.564,E2 -11598.564} C_VEL
LIN {X 0,Y 389.363,Z 452.124,A -85,B 0,C 180,E1 -11600.126,E2 -11600.126} C_VEL
LIN {X 0,Y 389.083,Z 458.4,A -85,B 0,C 180,E1 -11601.691,E2 -11601.691} C_VEL
LIN {X 0,Y 388.899,Z 463.373,A -85,B 0,C 180,E1 -11603.254,E2 -11603.254} C_VEL
LIN {X 0,Y 388.883,Z 467.196,A -85,B 0,C 180,E1 -11604.816,E2 -11604.816} C_VEL
LIN {X 0,Y 388.804,Z 469.145,A -85,B 0,C 180,E1 -11605.854,E2 -11605.854} C_VEL
LIN {X 0,Y 388.918,Z 470.681,A -85,B 0,C 180,E1 -11606.892,E2 -11606.892} C_VEL
LIN {X 0,Y 388.942,Z 471.744,A -85,B 0,C 180,E1 -11607.929,E2 -11607.929} C_VEL
LIN {X 0,Y 388.977,Z 472.391,A -85,B 0,C 180,E1 -11608.965,E2 -11608.965} C_VEL
LIN {X 0,Y 388.964,Z 472.634,A -85,B 0,C 180,E1 -11610,E2 -11610} C_VEL
LIN {X 0,Y 388.946,Z 472.474,A -85,B 0,C 180,E1 -11611.035,E2 -11611.035} C_VEL
LIN {X 0,Y 388.927,Z 471.867,A -85,B 0,C 180,E1 -11612.071,E2 -11612.071} C_VEL
LIN {X 0,Y 388.909,Z 470.849,A -85,B 0,C 180,E1 -11613.108,E2 -11613.108} C_VEL
LIN {X 0,Y 388.802,Z 469.416,A -85,B 0,C 180,E1 -11614.146,E2 -11614.146} C_VEL
LIN {X 0,Y 388.802,Z 466.104,A -85,B 0,C 180,E1 -11615.858,E2 -11615.858} C_VEL
LIN {X 0,Y 388.931,Z 462.41,A -85,B 0,C 180,E1 -11617.267,E2 -11617.267} C_VEL
LIN {X 0,Y 389.163,Z 456.283,A -85,B 0,C 180,E1 -11619.092,E2 -11619.092} C_VEL
LIN {X 0,Y 389.582,Z 449.57,A -85,B 0,C 180,E1 -11620.656,E2 -11620.656} C_VEL
LIN {X 0,Y 390.338,Z 441.286,A -85,B 0,C 180,E1 -11622.214,E2 -11622.214} C_VEL
LIN {X 0,Y 391.062,Z 432.877,A -85,B 0,C 180,E1 -11623.511,E2 -11623.511} C_VEL
LIN {X 0,Y 391.885,Z 422.667,A -85,B 0,C 180,E1 -11624.807,E2 -11624.807} C_VEL
LIN {X 0,Y 393.012,Z 411.23,A -85,B 0,C 180,E1 -11625.959,E2 -11625.959} C_VEL
LIN {X 0,Y 393.771,Z 400.157,A -85,B 0,C 180,E1 -11626.859,E2 -11626.859} C_VEL
LIN {X 0,Y 393.142,Z 388.076,A -85,B 0,C 180,E1 -11627.692,E2 -11627.692} C_VEL
LIN {X 0,Y 391.515,Z 374.438,A -85,B 0,C 180,E1 -11628.444,E2 -11628.444} C_VEL
LIN {X 0,Y 389.312,Z 362.314,A -85,B 0,C 180,E1 -11628.996,E2 -11628.996} C_VEL
LIN {X 0,Y 389.776,Z 352.782,A -85,B 0,C 180,E1 -11632.698,E2 -11632.698} C_VEL
LIN {X 0,Y 390.305,Z 344.05,A -85,B 0,C 180,E1 -11636.203,E2 -11636.203} C_VEL
LIN {X 0,Y 390.835,Z 337.206,A -85,B 0,C 180,E1 -11639.046,E2 -11639.046} C_VEL
LIN {X 0,Y 391.686,Z 329.054,A -85,B 0,C 180,E1 -11642.568,E2 -11642.568} C_VEL
LIN {X 0,Y 392.439,Z 322.484,A -85,B 0,C 180,E1 -11645.594,E2 -11645.594} C_VEL
LIN {X 0,Y 392.379,Z 318.617,A -85,B 0,C 180,E1 -11647.516,E2 -11647.516} C_VEL
LIN {X 0,Y 391.281,Z 312.293,A -85,B 0,C 180,E1 -11651.028,E2 -11651.028} C_VEL
LIN {X 0,Y 390.361,Z 307.597,A -85,B 0,C 180,E1 -11653.933,E2 -11653.933} C_VEL
LIN {X 0,Y 390.05,Z 305.908,A -85,B 0,C 180,E1 -11655.169,E2 -11655.169} C_VEL
LIN {X 0,Y 390.035,Z 305.907,A -85,B 0,C 180,E1 -11658.187,E2 -11658.187} C_VEL
LIN {X 0,Y 390.094,Z 305.9,A -85,B 0,C 180,E1 -11660.908,E2 -11660.908} C_VEL
LIN {X 0,Y 390.089,Z 305.895,A -85,B 0,C 180,E1 -11664.793,E2 -11664.793} C_VEL
LIN {X 0,Y 390.036,Z 305.902,A -85,B 0,C 180,E1 -11667.875,E2 -11667.875} C_VEL
LIN {X 0,Y 390.063,Z 305.899,A -85,B 0,C 180,E1 -11670.891,E2 -11670.891} C_VEL
LIN {X 0,Y 390.124,Z 305.892,A -85,B 0,C 180,E1 -11674.257,E2 -11674.257} C_VEL
LIN {X 0,Y 390.045,Z 305.898,A -85,B 0,C 180,E1 -11677.766,E2 -11677.766} C_VEL
LIN {X 0,Y 390.109,Z 305.894,A -85,B 0,C 180,E1 -11681.078,E2 -11681.078} C_VEL
LIN {X 0,Y 390.144,Z 305.886,A -85,B 0,C 180,E1 -11684.323,E2 -11684.323} C_VEL
LIN {X 0,Y 390.176,Z 305.885,A -85,B 0,C 180,E1 -11687.517,E2 -11687.517} C_VEL
LIN {X 0,Y 390.198,Z 305.882,A -85,B 0,C 180,E1 -11690.671,E2 -11690.671} C_VEL
LIN {X 0,Y 390.303,Z 305.868,A -85,B 0,C 180,E1 -11693.798,E2 -11693.798} C_VEL
LIN {X 0,Y 390.423,Z 305.854,A -85,B 0,C 180,E1 -11697.937,E2 -11697.937} C_VEL
LIN {X 0,Y 390.553,Z 305.839,A -85,B 0,C 180,E1 -11700,E2 -11700} C_VEL
LIN {X 0,Y 390.319,Z 305.868,A -85,B 0,C 180,E1 -11703.096,E2 -11703.096} C_VEL
LIN {X 0,Y 390.281,Z 305.871,A -85,B 0,C 180,E1 -11706.514,E2 -11706.514} C_VEL
LIN {X 0,Y 390.216,Z 305.881,A -85,B 0,C 180,E1 -11708.284,E2 -11708.284} C_VEL
LIN {X 0,Y 389.962,Z 305.916,A -85,B 0,C 180,E1 -11710.383,E2 -11710.383} C_VEL
LIN {X 0,Y 389.885,Z 308.012,A -85,B 0,C 180,E1 -11713.244,E2 -11713.244} C_VEL
LIN {X 0,Y 389.727,Z 310.993,A -85,B 0,C 180,E1 -11716.77,E2 -11716.77} C_VEL
LIN {X 0,Y 389.604,Z 313.095,A -85,B 0,C 180,E1 -11719.186,E2 -11719.186} C_VEL
LIN {X 0,Y 393.881,Z 326.657,A -85,B 0,C 180,E1 -11719.993,E2 -11719.993} C_VEL
LIN {X 0,Y 396.008,Z 335.731,A -85,B 0,C 180,E1 -11720.626,E2 -11720.626} C_VEL
LIN {X 0,Y 395.233,Z 348.622,A -85,B 0,C 180,E1 -11721.515,E2 -11721.515} C_VEL
LIN {X 0,Y 394.237,Z 360.388,A -85,B 0,C 180,E1 -11722.578,E2 -11722.578} C_VEL
LIN {X 0,Y 393.3,Z 371.344,A -85,B 0,C 180,E1 -11723.831,E2 -11723.831} C_VEL
LIN {X 0,Y 392.389,Z 380.754,A -85,B 0,C 180,E1 -11725.175,E2 -11725.175} C_VEL
LIN {X 0,Y 391.556,Z 389.151,A -85,B 0,C 180,E1 -11726.662,E2 -11726.662} C_VEL
LIN {X 0,Y 390.795,Z 396.219,A -85,B 0,C 180,E1 -11728.21,E2 -11728.21} C_VEL
LIN {X 0,Y 390.26,Z 401.34,A -85,B 0,C 180,E1 -11729.607,E2 -11729.607} C_VEL
LIN {X 0,Y 389.697,Z 406.809,A -85,B 0,C 180,E1 -11731.534,E2 -11731.534} C_VEL
LIN {X 0,Y 389.454,Z 409.459,A -85,B 0,C 180,E1 -11732.777,E2 -11732.777} C_VEL
LIN {X 0,Y 389.199,Z 411.491,A -85,B 0,C 180,E1 -11734.041,E2 -11734.041} C_VEL
LIN {X 0,Y 388.965,Z 413.161,A -85,B 0,C 180,E1 -11735.601,E2 -11735.601} C_VEL
LIN {X 0,Y 388.846,Z 413.933,A -85,B 0,C 180,E1 -11737.32,E2 -11737.32} C_VEL
LIN {X 0,Y 388.865,Z 413.506,A -85,B 0,C 180,E1 -11739.239,E2 -11739.239} C_VEL
LIN {X 0,Y 388.939,Z 412.338,A -85,B 0,C 180,E1 -11740.63,E2 -11740.63} C_VEL
LIN {X 0,Y 389.129,Z 410.089,A -85,B 0,C 180,E1 -11742.226,E2 -11742.226} C_VEL
LIN {X 0,Y 389.438,Z 406.882,A -85,B 0,C 180,E1 -11743.791,E2 -11743.791} C_VEL
LIN {X 0,Y 389.81,Z 401.584,A -85,B 0,C 180,E1 -11745.681,E2 -11745.681} C_VEL
LIN {X 0,Y 390.178,Z 396.264,A -85,B 0,C 180,E1 -11747.145,E2 -11747.145} C_VEL
LIN {X 0,Y 390.806,Z 388.635,A -85,B 0,C 180,E1 -11748.819,E2 -11748.819} C_VEL
LIN {X 0,Y 391.548,Z 379.754,A -85,B 0,C 180,E1 -11750.367,E2 -11750.367} C_VEL
LIN {X 0,Y 392.256,Z 371.087,A -85,B 0,C 180,E1 -11751.599,E2 -11751.599} C_VEL
LIN {X 0,Y 393.061,Z 360.74,A -85,B 0,C 180,E1 -11752.8,E2 -11752.8} C_VEL
LIN {X 0,Y 393.85,Z 348.525,A -85,B 0,C 180,E1 -11753.923,E2 -11753.923} C_VEL
LIN {X 0,Y 394.637,Z 336.603,A -85,B 0,C 180,E1 -11754.771,E2 -11754.771} C_VEL
LIN {X 0,Y 394.678,Z 332.857,A -85,B 0,C 180,E1 -11754.997,E2 -11754.997} C_VEL
LIN {X 0,Y 391.779,Z 320.33,A -85,B 0,C 180,E1 -11755.748,E2 -11755.748} C_VEL
LIN {X 0,Y 389.187,Z 310.303,A -85,B 0,C 180,E1 -11756.219,E2 -11756.219} C_VEL
LIN {X 0,Y 389.222,Z 306.828,A -85,B 0,C 180,E1 -11759.63,E2 -11759.63} C_VEL
LIN {X 0,Y 389.293,Z 305.996,A -85,B 0,C 180,E1 -11760.827,E2 -11760.827} C_VEL
LIN {X 0,Y 389.785,Z 305.931,A -85,B 0,C 180,E1 -11764.359,E2 -11764.359} C_VEL
LIN {X 0,Y 390.011,Z 305.904,A -85,B 0,C 180,E1 -11767.764,E2 -11767.764} C_VEL
LIN {X 0,Y 390.103,Z 305.895,A -85,B 0,C 180,E1 -11771.078,E2 -11771.078} C_VEL
LIN {X 0,Y 390.14,Z 305.886,A -85,B 0,C 180,E1 -11774.323,E2 -11774.323} C_VEL
LIN {X 0,Y 390.172,Z 305.883,A -85,B 0,C 180,E1 -11777.517,E2 -11777.517} C_VEL
LIN {X 0,Y 390.205,Z 305.881,A -85,B 0,C 180,E1 -11780.671,E2 -11780.671} C_VEL
LIN {X 0,Y 390.3,Z 305.866,A -85,B 0,C 180,E1 -11783.798,E2 -11783.798} C_VEL
LIN {X 0,Y 390.419,Z 305.852,A -85,B 0,C 180,E1 -11787.937,E2 -11787.937} C_VEL
LIN {X 0,Y 390.549,Z 305.835,A -85,B 0,C 180,E1 -11790,E2 -11790} C_VEL
LIN {X 0,Y 390.316,Z 305.866,A -85,B 0,C 180,E1 -11793.097,E2 -11793.097} C_VEL
LIN {X 0,Y 390.3,Z 305.869,A -85,B 0,C 180,E1 -11796.202,E2 -11796.202} C_VEL
LIN {X 0,Y 390.205,Z 305.878,A -85,B 0,C 180,E1 -11799.329,E2 -11799.329} C_VEL
LIN {X 0,Y 390.195,Z 305.879,A -85,B 0,C 180,E1 -11803.439,E2 -11803.439} C_VEL
LIN {X 0,Y 390.15,Z 305.885,A -85,B 0,C 180,E1 -11807.308,E2 -11807.308} C_VEL
LIN {X 0,Y 390.098,Z 305.89,A -85,B 0,C 180,E1 -11808.446,E2 -11808.446} C_VEL
LIN {X 0,Y 389.422,Z 305.976,A -85,B 0,C 180,E1 -11809.308,E2 -11809.308} C_VEL
LIN {X 0,Y 386.538,Z 306.338,A -85,B 0,C 180,E1 -11810.708,E2 -11810.708} C_VEL
LIN {X 0,Y 384.111,Z 306.64,A -85,B 0,C 180,E1 -11811.84,E2 -11811.84} C_VEL
LIN {X 0,Y 383.087,Z 306.767,A -85,B 0,C 180,E1 -11812.715,E2 -11812.715} C_VEL
LIN {X 0,Y 383.014,Z 306.774,A -85,B 0,C 180,E1 -11813.012,E2 -11813.012} C_VEL
LIN {X 0,Y 383.081,Z 306.769,A -85,B 0,C 180,E1 -11816.123,E2 -11816.123} C_VEL
LIN {X 0,Y 383.041,Z 306.773,A -85,B 0,C 180,E1 -11818.493,E2 -11818.493} C_VEL
LIN {X 0,Y 383.011,Z 306.778,A -85,B 0,C 180,E1 -11822.15,E2 -11822.15} C_VEL
LIN {X 0,Y 383.019,Z 306.774,A -85,B 0,C 180,E1 -11824.668,E2 -11824.668} C_VEL
LIN {X 0,Y 383.001,Z 306.779,A -85,B 0,C 180,E1 -11827.904,E2 -11827.904} C_VEL
LIN {X 0,Y 382.985,Z 306.778,A -85,B 0,C 180,E1 -11831.348,E2 -11831.348} C_VEL
LIN {X 0,Y 382.997,Z 306.777,A -85,B 0,C 180,E1 -11834.304,E2 -11834.304} C_VEL
LIN {X 0,Y 383.012,Z 306.775,A -85,B 0,C 180,E1 -11837.24,E2 -11837.24} C_VEL
LIN {X 0,Y 383.018,Z 306.774,A -85,B 0,C 180,E1 -11840.414,E2 -11840.414} C_VEL
LIN {X 0,Y 383.027,Z 306.774,A -85,B 0,C 180,E1 -11844.045,E2 -11844.045} C_VEL
LIN {X 0,Y 382.989,Z 306.78,A -85,B 0,C 180,E1 -11847.578,E2 -11847.578} C_VEL
LIN {X 0,Y 382.995,Z 306.776,A -85,B 0,C 180,E1 -11850.3,E2 -11850.3} C_VEL
LIN {X 0,Y 383.059,Z 306.768,A -85,B 0,C 180,E1 -11852.698,E2 -11852.698} C_VEL
LIN {X 0,Y 383.052,Z 306.771,A -85,B 0,C 180,E1 -11855.04,E2 -11855.04} C_VEL
LIN {X 0,Y 382.996,Z 306.776,A -85,B 0,C 180,E1 -11858.469,E2 -11858.469} C_VEL
LIN {X 0,Y 383.056,Z 306.769,A -85,B 0,C 180,E1 -11861.826,E2 -11861.826} C_VEL
LIN {X 0,Y 383.114,Z 306.765,A -85,B 0,C 180,E1 -11865.119,E2 -11865.119} C_VEL
LIN {X 0,Y 383.101,Z 306.763,A -85,B 0,C 180,E1 -11868.358,E2 -11868.358} C_VEL
LIN {X 0,Y 383.233,Z 306.746,A -85,B 0,C 180,E1 -11872.013,E2 -11872.013} C_VEL
LIN {X 0,Y 383.2,Z 306.754,A -85,B 0,C 180,E1 -11874.739,E2 -11874.739} C_VEL
LIN {X 0,Y 383.388,Z 306.726,A -85,B 0,C 180,E1 -11877.899,E2 -11877.899} C_VEL
LIN {X 0,Y 383.52,Z 306.711,A -85,B 0,C 180,E1 -11880,E2 -11880} C_VEL
LIN {X 0,Y 383.216,Z 306.752,A -85,B 0,C 180,E1 -11883.154,E2 -11883.154} C_VEL
LIN {X 0,Y 383.259,Z 306.744,A -85,B 0,C 180,E1 -11886.317,E2 -11886.317} C_VEL
LIN {X 0,Y 383.148,Z 306.756,A -85,B 0,C 180,E1 -11889.502,E2 -11889.502} C_VEL
LIN {X 0,Y 383.13,Z 306.758,A -85,B 0,C 180,E1 -11893.536,E2 -11893.536} C_VEL
LIN {X 0,Y 383.098,Z 306.764,A -85,B 0,C 180,E1 -11897.069,E2 -11897.069} C_VEL
LIN {X 0,Y 383.033,Z 306.775,A -85,B 0,C 180,E1 -11900.647,E2 -11900.647} C_VEL
LIN {X 0,Y 383.021,Z 306.774,A -85,B 0,C 180,E1 -11903.808,E2 -11903.808} C_VEL
LIN {X 0,Y 383.022,Z 306.773,A -85,B 0,C 180,E1 -11907.305,E2 -11907.305} C_VEL
LIN {X 0,Y 382.986,Z 306.778,A -85,B 0,C 180,E1 -11910.919,E2 -11910.919} C_VEL
LIN {X 0,Y 383.022,Z 306.774,A -85,B 0,C 180,E1 -11914.668,E2 -11914.668} C_VEL
LIN {X 0,Y 383.001,Z 306.779,A -85,B 0,C 180,E1 -11917.903,E2 -11917.903} C_VEL
LIN {X 0,Y 382.984,Z 306.778,A -85,B 0,C 180,E1 -11921.348,E2 -11921.348} C_VEL
LIN {X 0,Y 382.998,Z 306.778,A -85,B 0,C 180,E1 -11924.303,E2 -11924.303} C_VEL
LIN {X 0,Y 383.067,Z 306.921,A -85,B 0,C 180,E1 -11926.353,E2 -11926.353} C_VEL
LIN {X 0,Y 384.431,Z 314.412,A -85,B 0,C 180,E1 -11930.159,E2 -11930.159} C_VEL
LIN {X 0,Y 385.418,Z 320.324,A -85,B 0,C 180,E1 -11933.005,E2 -11933.005} C_VEL
LIN {X 0,Y 385.199,Z 325.207,A -85,B 0,C 180,E1 -11935.188,E2 -11935.188} C_VEL
LIN {X 0,Y 384.385,Z 333.07,A -85,B 0,C 180,E1 -11938.595,E2 -11938.595} C_VEL
LIN {X 0,Y 383.668,Z 341.553,A -85,B 0,C 180,E1 -11942.153,E2 -11942.153} C_VEL
LIN {X 0,Y 382.992,Z 349.979,A -85,B 0,C 180,E1 -11945.614,E2 -11945.614} C_VEL
LIN {X 0,Y 382.464,Z 358.398,A -85,B 0,C 180,E1 -11949.003,E2 -11949.003} C_VEL
LIN {X 0,Y 382.238,Z 364.469,A -85,B 0,C 180,E1 -11951.404,E2 -11951.404} C_VEL
LIN {X 0,Y 384.319,Z 379.569,A -85,B 0,C 180,E1 -11952.028,E2 -11952.028} C_VEL
LIN {X 0,Y 385.769,Z 393.275,A -85,B 0,C 180,E1 -11952.814,E2 -11952.814} C_VEL
LIN {X 0,Y 386.199,Z 402.599,A -85,B 0,C 180,E1 -11953.48,E2 -11953.48} C_VEL
LIN {X 0,Y 385.199,Z 414.868,A -85,B 0,C 180,E1 -11954.524,E2 -11954.524} C_VEL
LIN {X 0,Y 384.335,Z 424.966,A -85,B 0,C 180,E1 -11955.613,E2 -11955.613} C_VEL
LIN {X 0,Y 383.51,Z 435.505,A -85,B 0,C 180,E1 -11957.027,E2 -11957.027} C_VEL
LIN {X 0,Y 382.898,Z 443.55,A -85,B 0,C 180,E1 -11958.352,E2 -11958.352} C_VEL
LIN {X 0,Y 382.312,Z 451.435,A -85,B 0,C 180,E1 -11959.942,E2 -11959.942} C_VEL
LIN {X 0,Y 382.006,Z 457.74,A -85,B 0,C 180,E1 -11961.536,E2 -11961.536} C_VEL
LIN {X 0,Y 381.831,Z 462.743,A -85,B 0,C 180,E1 -11963.129,E2 -11963.129} C_VEL
LIN {X 0,Y 381.791,Z 466.589,A -85,B 0,C 180,E1 -11964.719,E2 -11964.719} C_VEL
LIN {X 0,Y 381.728,Z 468.552,A -85,B 0,C 180,E1 -11965.777,E2 -11965.777} C_VEL
LIN {X 0,Y 381.821,Z 470.099,A -85,B 0,C 180,E1 -11966.835,E2 -11966.835} C_VEL
LIN {X 0,Y 381.871,Z 471.182,A -85,B 0,C 180,E1 -11967.891,E2 -11967.891} C_VEL
LIN {X 0,Y 381.896,Z 471.837,A -85,B 0,C 180,E1 -11968.946,E2 -11968.946} C_VEL
LIN {X 0,Y 381.914,Z 472.09,A -85,B 0,C 180,E1 -11970,E2 -11970} C_VEL
LIN {X 0,Y 381.867,Z 471.939,A -85,B 0,C 180,E1 -11971.055,E2 -11971.055} C_VEL
LIN {X 0,Y 381.858,Z 471.348,A -85,B 0,C 180,E1 -11972.11,E2 -11972.11} C_VEL
LIN {X 0,Y 381.809,Z 470.335,A -85,B 0,C 180,E1 -11973.166,E2 -11973.166} C_VEL
LIN {X 0,Y 381.723,Z 468.914,A -85,B 0,C 180,E1 -11974.223,E2 -11974.223} C_VEL
LIN {X 0,Y 381.756,Z 467.08,A -85,B 0,C 180,E1 -11975.282,E2 -11975.282} C_VEL
LIN {X 0,Y 381.784,Z 463.433,A -85,B 0,C 180,E1 -11976.872,E2 -11976.872} C_VEL
LIN {X 0,Y 381.993,Z 458.688,A -85,B 0,C 180,E1 -11978.464,E2 -11978.464} C_VEL
LIN {X 0,Y 382.379,Z 451.55,A -85,B 0,C 180,E1 -11980.323,E2 -11980.323} C_VEL
LIN {X 0,Y 383.06,Z 443.877,A -85,B 0,C 180,E1 -11981.912,E2 -11981.912} C_VEL
LIN {X 0,Y 383.739,Z 436.098,A -85,B 0,C 180,E1 -11983.234,E2 -11983.234} C_VEL
LIN {X 0,Y 384.572,Z 426.633,A -85,B 0,C 180,E1 -11984.566,E2 -11984.566} C_VEL
LIN {X 0,Y 385.728,Z 415.141,A -85,B 0,C 180,E1 -11985.861,E2 -11985.861} C_VEL
LIN {X 0,Y 386.848,Z 403.595,A -85,B 0,C 180,E1 -11986.899,E2 -11986.899} C_VEL
LIN {X 0,Y 386.466,Z 391.775,A -85,B 0,C 180,E1 -11987.793,E2 -11987.793} C_VEL
LIN {X 0,Y 385.28,Z 378.759,A -85,B 0,C 180,E1 -11988.588,E2 -11988.588} C_VEL
LIN {X 0,Y 382.836,Z 364.807,A -85,B 0,C 180,E1 -11989.277,E2 -11989.277} C_VEL
LIN {X 0,Y 382.271,Z 361.767,A -85,B 0,C 180,E1 -11989.395,E2 -11989.395} C_VEL
LIN {X 0,Y 382.706,Z 353.502,A -85,B 0,C 180,E1 -11992.684,E2 -11992.684} C_VEL
LIN {X 0,Y 383.317,Z 343.755,A -85,B 0,C 180,E1 -11996.693,E2 -11996.693} C_VEL
LIN {X 0,Y 383.895,Z 336.917,A -85,B 0,C 180,E1 -11999.623,E2 -11999.623} C_VEL
LIN {X 0,Y 384.823,Z 328.876,A -85,B 0,C 180,E1 -12003.223,E2 -12003.223} C_VEL
LIN {X 0,Y 385.477,Z 323.635,A -85,B 0,C 180,E1 -12005.692,E2 -12005.692} C_VEL
LIN {X 0,Y 385.541,Z 321.032,A -85,B 0,C 180,E1 -12006.982,E2 -12006.982} C_VEL
LIN {X 0,Y 384.68,Z 315.79,A -85,B 0,C 180,E1 -12009.885,E2 -12009.885} C_VEL
LIN {X 0,Y 383.793,Z 310.803,A -85,B 0,C 180,E1 -12012.905,E2 -12012.905} C_VEL
LIN {X 0,Y 382.999,Z 306.784,A -85,B 0,C 180,E1 -12015.697,E2 -12015.697} C_VEL
LIN {X 0,Y 382.992,Z 306.784,A -85,B 0,C 180,E1 -12018.796,E2 -12018.796} C_VEL
LIN {X 0,Y 383.004,Z 306.78,A -85,B 0,C 180,E1 -12022.096,E2 -12022.096} C_VEL
LIN {X 0,Y 383.022,Z 306.774,A -85,B 0,C 180,E1 -12025.332,E2 -12025.332} C_VEL
LIN {X 0,Y 382.987,Z 306.781,A -85,B 0,C 180,E1 -12029.082,E2 -12029.082} C_VEL
LIN {X 0,Y 383.061,Z 306.771,A -85,B 0,C 180,E1 -12032.698,E2 -12032.698} C_VEL
LIN {X 0,Y 383.057,Z 306.77,A -85,B 0,C 180,E1 -12035.04,E2 -12035.04} C_VEL
LIN {X 0,Y 382.998,Z 306.779,A -85,B 0,C 180,E1 -12038.469,E2 -12038.469} C_VEL
LIN {X 0,Y 383.093,Z 306.765,A -85,B 0,C 180,E1 -12041.828,E2 -12041.828} C_VEL
LIN {X 0,Y 383.115,Z 306.763,A -85,B 0,C 180,E1 -12045.118,E2 -12045.118} C_VEL
LIN {X 0,Y 383.102,Z 306.765,A -85,B 0,C 180,E1 -12048.358,E2 -12048.358} C_VEL
LIN {X 0,Y 383.224,Z 306.751,A -85,B 0,C 180,E1 -12052.022,E2 -12052.022} C_VEL
LIN {X 0,Y 383.192,Z 306.755,A -85,B 0,C 180,E1 -12054.738,E2 -12054.738} C_VEL
LIN {X 0,Y 383.39,Z 306.73,A -85,B 0,C 180,E1 -12057.899,E2 -12057.899} C_VEL
LIN {X 0,Y 383.523,Z 306.715,A -85,B 0,C 180,E1 -12060,E2 -12060} C_VEL
LIN {X 0,Y 383.256,Z 306.747,A -85,B 0,C 180,E1 -12063.153,E2 -12063.153} C_VEL
LIN {X 0,Y 383.245,Z 306.748,A -85,B 0,C 180,E1 -12066.503,E2 -12066.503} C_VEL
LIN {X 0,Y 383.157,Z 306.761,A -85,B 0,C 180,E1 -12068.438,E2 -12068.438} C_VEL
LIN {X 0,Y 382.92,Z 306.928,A -85,B 0,C 180,E1 -12070.576,E2 -12070.576} C_VEL
LIN {X 0,Y 382.814,Z 309.542,A -85,B 0,C 180,E1 -12073.808,E2 -12073.808} C_VEL
LIN {X 0,Y 382.653,Z 312.401,A -85,B 0,C 180,E1 -12077.241,E2 -12077.241} C_VEL
LIN {X 0,Y 382.579,Z 313.699,A -85,B 0,C 180,E1 -12078.752,E2 -12078.752} C_VEL
LIN {X 0,Y 387.042,Z 327.655,A -85,B 0,C 180,E1 -12079.629,E2 -12079.629} C_VEL
LIN {X 0,Y 389.126,Z 335.598,A -85,B 0,C 180,E1 -12080.207,E2 -12080.207} C_VEL
LIN {X 0,Y 389.224,Z 339.658,A -85,B 0,C 180,E1 -12080.478,E2 -12080.478} C_VEL
LIN {X 0,Y 388.364,Z 351.411,A -85,B 0,C 180,E1 -12081.358,E2 -12081.358} C_VEL
LIN {X 0,Y 387.414,Z 362.295,A -85,B 0,C 180,E1 -12082.393,E2 -12082.393} C_VEL
LIN {X 0,Y 386.486,Z 372.331,A -85,B 0,C 180,E1 -12083.582,E2 -12083.582} C_VEL
LIN {X 0,Y 385.651,Z 380.604,A -85,B 0,C 180,E1 -12084.781,E2 -12084.781} C_VEL
LIN {X 0,Y 384.789,Z 388.734,A -85,B 0,C 180,E1 -12086.219,E2 -12086.219} C_VEL
LIN {X 0,Y 383.935,Z 396.096,A -85,B 0,C 180,E1 -12087.825,E2 -12087.825} C_VEL
LIN {X 0,Y 383.296,Z 401.766,A -85,B 0,C 180,E1 -12089.372,E2 -12089.372} C_VEL
LIN {X 0,Y 382.826,Z 406.282,A -85,B 0,C 180,E1 -12090.933,E2 -12090.933} C_VEL
LIN {X 0,Y 382.375,Z 410.392,A -85,B 0,C 180,E1 -12092.843,E2 -12092.843} C_VEL
LIN {X 0,Y 382.024,Z 413.044,A -85,B 0,C 180,E1 -12094.771,E2 -12094.771} C_VEL
LIN {X 0,Y 381.869,Z 414.1,A -85,B 0,C 180,E1 -12096.081,E2 -12096.081} C_VEL
LIN {X 0,Y 381.769,Z 414.515,A -85,B 0,C 180,E1 -12097.665,E2 -12097.665} C_VEL
LIN {X 0,Y 381.805,Z 413.971,A -85,B 0,C 180,E1 -12099.366,E2 -12099.366} C_VEL
LIN {X 0,Y 381.954,Z 411.821,A -85,B 0,C 180,E1 -12101.483,E2 -12101.483} C_VEL
LIN {X 0,Y 382.196,Z 409.522,A -85,B 0,C 180,E1 -12102.873,E2 -12102.873} C_VEL
LIN {X 0,Y 382.429,Z 406.355,A -85,B 0,C 180,E1 -12104.294,E2 -12104.294} C_VEL
LIN {X 0,Y 382.87,Z 401.072,A -85,B 0,C 180,E1 -12106.093,E2 -12106.093} C_VEL
LIN {X 0,Y 383.393,Z 393.993,A -85,B 0,C 180,E1 -12107.936,E2 -12107.936} C_VEL
LIN {X 0,Y 384.063,Z 386.467,A -85,B 0,C 180,E1 -12109.488,E2 -12109.488} C_VEL
LIN {X 0,Y 384.813,Z 377.697,A -85,B 0,C 180,E1 -12110.943,E2 -12110.943} C_VEL
LIN {X 0,Y 385.61,Z 368.36,A -85,B 0,C 180,E1 -12112.207,E2 -12112.207} C_VEL
LIN {X 0,Y 386.413,Z 357.766,A -85,B 0,C 180,E1 -12113.377,E2 -12113.377} C_VEL
LIN {X 0,Y 387.122,Z 347.089,A -85,B 0,C 180,E1 -12114.323,E2 -12114.323} C_VEL
LIN {X 0,Y 387.855,Z 335.151,A -85,B 0,C 180,E1 -12115.145,E2 -12115.145} C_VEL
LIN {X 0,Y 385.977,Z 325.835,A -85,B 0,C 180,E1 -12115.749,E2 -12115.749} C_VEL
LIN {X 0,Y 382.468,Z 312.333,A -85,B 0,C 180,E1 -12116.449,E2 -12116.449} C_VEL
LIN {X 0,Y 382.139,Z 310.772,A -85,B 0,C 180,E1 -12116.533,E2 -12116.533} C_VEL
LIN {X 0,Y 382.193,Z 307.016,A -85,B 0,C 180,E1 -12120.232,E2 -12120.232} C_VEL
LIN {X 0,Y 382.498,Z 306.84,A -85,B 0,C 180,E1 -12122.655,E2 -12122.655} C_VEL
LIN {X 0,Y 382.764,Z 306.809,A -85,B 0,C 180,E1 -12125.019,E2 -12125.019} C_VEL
LIN {X 0,Y 382.945,Z 306.786,A -85,B 0,C 180,E1 -12127.331,E2 -12127.331} C_VEL
LIN {X 0,Y 383.059,Z 306.769,A -85,B 0,C 180,E1 -12130.716,E2 -12130.716} C_VEL
LIN {X 0,Y 383.081,Z 306.764,A -85,B 0,C 180,E1 -12134.027,E2 -12134.027} C_VEL
LIN {X 0,Y 383.137,Z 306.761,A -85,B 0,C 180,E1 -12137.284,E2 -12137.284} C_VEL
LIN {X 0,Y 383.152,Z 306.759,A -85,B 0,C 180,E1 -12140.498,E2 -12140.498} C_VEL
LIN {X 0,Y 383.256,Z 306.744,A -85,B 0,C 180,E1 -12143.683,E2 -12143.683} C_VEL
LIN {X 0,Y 383.386,Z 306.727,A -85,B 0,C 180,E1 -12147.899,E2 -12147.899} C_VEL
LIN {X 0,Y 383.519,Z 306.711,A -85,B 0,C 180,E1 -12150,E2 -12150} C_VEL
LIN {X 0,Y 383.252,Z 306.745,A -85,B 0,C 180,E1 -12153.154,E2 -12153.154} C_VEL
LIN {X 0,Y 383.256,Z 306.747,A -85,B 0,C 180,E1 -12156.317,E2 -12156.317} C_VEL
LIN {X 0,Y 383.151,Z 306.756,A -85,B 0,C 180,E1 -12159.502,E2 -12159.502} C_VEL
LIN {X 0,Y 383.126,Z 306.76,A -85,B 0,C 180,E1 -12163.536,E2 -12163.536} C_VEL
LIN {X 0,Y 383.095,Z 306.763,A -85,B 0,C 180,E1 -12167.455,E2 -12167.455} C_VEL
LIN {X 0,Y 383.03,Z 306.774,A -85,B 0,C 180,E1 -12170.647,E2 -12170.647} C_VEL
LIN {X 0,Y 383.014,Z 306.774,A -85,B 0,C 180,E1 -12173.012,E2 -12173.012} C_VEL
LIN {X 0,Y 382.369,Z 306.857,A -85,B 0,C 180,E1 -12173.89,E2 -12173.89} C_VEL
LIN {X 0,Y 379.512,Z 307.21,A -85,B 0,C 180,E1 -12175.318,E2 -12175.318} C_VEL
LIN {X 0,Y 377.089,Z 307.515,A -85,B 0,C 180,E1 -12176.473,E2 -12176.473} C_VEL
LIN {X 0,Y 376.064,Z 307.639,A -85,B 0,C 180,E1 -12177.366,E2 -12177.366} C_VEL
LIN {X 0,Y 375.99,Z 307.649,A -85,B 0,C 180,E1 -12177.668,E2 -12177.668} C_VEL
LIN {X 0,Y 375.959,Z 307.653,A -85,B 0,C 180,E1 -12181.562,E2 -12181.562} C_VEL
LIN {X 0,Y 375.958,Z 307.653,A -85,B 0,C 180,E1 -12185.416,E2 -12185.416} C_VEL
LIN {X 0,Y 375.975,Z 307.653,A -85,B 0,C 180,E1 -12188.271,E2 -12188.271} C_VEL
LIN {X 0,Y 375.936,Z 307.658,A -85,B 0,C 180,E1 -12191.601,E2 -12191.601} C_VEL
LIN {X 0,Y 375.929,Z 307.657,A -85,B 0,C 180,E1 -12195.269,E2 -12195.269} C_VEL
LIN {X 0,Y 375.937,Z 307.656,A -85,B 0,C 180,E1 -12198.399,E2 -12198.399} C_VEL
LIN {X 0,Y 375.977,Z 307.654,A -85,B 0,C 180,E1 -12201.73,E2 -12201.73} C_VEL
LIN {X 0,Y 375.982,Z 307.652,A -85,B 0,C 180,E1 -12205.333,E2 -12205.333} C_VEL
LIN {X 0,Y 375.96,Z 307.652,A -85,B 0,C 180,E1 -12208.438,E2 -12208.438} C_VEL
LIN {X 0,Y 375.999,Z 307.648,A -85,B 0,C 180,E1 -12212.142,E2 -12212.142} C_VEL
LIN {X 0,Y 376.007,Z 307.646,A -85,B 0,C 180,E1 -12214.539,E2 -12214.539} C_VEL
LIN {X 0,Y 375.96,Z 307.652,A -85,B 0,C 180,E1 -12218.046,E2 -12218.046} C_VEL
LIN {X 0,Y 376.006,Z 307.65,A -85,B 0,C 180,E1 -12221.473,E2 -12221.473} C_VEL
LIN {X 0,Y 376.062,Z 307.642,A -85,B 0,C 180,E1 -12224.833,E2 -12224.833} C_VEL
LIN {X 0,Y 376.054,Z 307.64,A -85,B 0,C 180,E1 -12228.137,E2 -12228.137} C_VEL
LIN {X 0,Y 376.205,Z 307.622,A -85,B 0,C 180,E1 -12231.938,E2 -12231.938} C_VEL
LIN {X 0,Y 376.172,Z 307.628,A -85,B 0,C 180,E1 -12234.64,E2 -12234.64} C_VEL
LIN {X 0,Y 376.354,Z 307.602,A -85,B 0,C 180,E1 -12237.86,E2 -12237.86} C_VEL
LIN {X 0,Y 376.49,Z 307.586,A -85,B 0,C 180,E1 -12240,E2 -12240} C_VEL
LIN {X 0,Y 376.349,Z 307.604,A -85,B 0,C 180,E1 -12242.141,E2 -12242.141} C_VEL
LIN {X 0,Y 376.217,Z 307.623,A -85,B 0,C 180,E1 -12246.436,E2 -12246.436} C_VEL
LIN {X 0,Y 376.118,Z 307.632,A -85,B 0,C 180,E1 -12249.682,E2 -12249.682} C_VEL
LIN {X 0,Y 376.094,Z 307.635,A -85,B 0,C 180,E1 -12253.658,E2 -12253.658} C_VEL
LIN {X 0,Y 376.036,Z 307.642,A -85,B 0,C 180,E1 -12257.4,E2 -12257.4} C_VEL
LIN {X 0,Y 375.982,Z 307.651,A -85,B 0,C 180,E1 -12260.832,E2 -12260.832} C_VEL
LIN {X 0,Y 375.981,Z 307.653,A -85,B 0,C 180,E1 -12264.283,E2 -12264.283} C_VEL
LIN {X 0,Y 375.968,Z 307.654,A -85,B 0,C 180,E1 -12266.656,E2 -12266.656} C_VEL
LIN {X 0,Y 375.966,Z 307.655,A -85,B 0,C 180,E1 -12270.313,E2 -12270.313} C_VEL
LIN {X 0,Y 375.966,Z 307.656,A -85,B 0,C 180,E1 -12274.111,E2 -12274.111} C_VEL
LIN {X 0,Y 375.956,Z 307.653,A -85,B 0,C 180,E1 -12276.741,E2 -12276.741} C_VEL
LIN {X 0,Y 375.99,Z 307.652,A -85,B 0,C 180,E1 -12279.97,E2 -12279.97} C_VEL
LIN {X 0,Y 375.932,Z 307.659,A -85,B 0,C 180,E1 -12283.766,E2 -12283.766} C_VEL
LIN {X 0,Y 376.001,Z 307.725,A -85,B 0,C 180,E1 -12286.014,E2 -12286.014} C_VEL
LIN {X 0,Y 377.341,Z 314.973,A -85,B 0,C 180,E1 -12289.785,E2 -12289.785} C_VEL
LIN {X 0,Y 378.412,Z 321.506,A -85,B 0,C 180,E1 -12292.998,E2 -12292.998} C_VEL
LIN {X 0,Y 378.276,Z 325.507,A -85,B 0,C 180,E1 -12294.833,E2 -12294.833} C_VEL
LIN {X 0,Y 377.335,Z 333.958,A -85,B 0,C 180,E1 -12298.566,E2 -12298.566} C_VEL
LIN {X 0,Y 376.684,Z 341.301,A -85,B 0,C 180,E1 -12301.721,E2 -12301.721} C_VEL
LIN {X 0,Y 375.994,Z 349.435,A -85,B 0,C 180,E1 -12305.13,E2 -12305.13} C_VEL
LIN {X 0,Y 375.458,Z 357.81,A -85,B 0,C 180,E1 -12308.592,E2 -12308.592} C_VEL
LIN {X 0,Y 375.171,Z 364.011,A -85,B 0,C 180,E1 -12311.111,E2 -12311.111} C_VEL
LIN {X 0,Y 377.152,Z 377.881,A -85,B 0,C 180,E1 -12311.676,E2 -12311.676} C_VEL
LIN {X 0,Y 378.573,Z 391.224,A -85,B 0,C 180,E1 -12312.436,E2 -12312.436} C_VEL
LIN {X 0,Y 379.291,Z 401.421,A -85,B 0,C 180,E1 -12313.171,E2 -12313.171} C_VEL
LIN {X 0,Y 378.301,Z 413.816,A -85,B 0,C 180,E1 -12314.234,E2 -12314.234} C_VEL
LIN {X 0,Y 377.304,Z 424.992,A -85,B 0,C 180,E1 -12315.462,E2 -12315.462} C_VEL
LIN {X 0,Y 376.561,Z 434.651,A -85,B 0,C 180,E1 -12316.784,E2 -12316.784} C_VEL
LIN {X 0,Y 375.899,Z 442.752,A -85,B 0,C 180,E1 -12318.132,E2 -12318.132} C_VEL
LIN {X 0,Y 375.249,Z 450.7,A -85,B 0,C 180,E1 -12319.751,E2 -12319.751} C_VEL
LIN {X 0,Y 374.944,Z 457.052,A -85,B 0,C 180,E1 -12321.376,E2 -12321.376} C_VEL
LIN {X 0,Y 374.75,Z 462.089,A -85,B 0,C 180,E1 -12322.998,E2 -12322.998} C_VEL
LIN {X 0,Y 374.702,Z 465.966,A -85,B 0,C 180,E1 -12324.619,E2 -12324.619} C_VEL
LIN {X 0,Y 374.653,Z 467.943,A -85,B 0,C 180,E1 -12325.697,E2 -12325.697} C_VEL
LIN {X 0,Y 374.727,Z 469.502,A -85,B 0,C 180,E1 -12326.775,E2 -12326.775} C_VEL
LIN {X 0,Y 374.801,Z 470.612,A -85,B 0,C 180,E1 -12327.851,E2 -12327.851} C_VEL
LIN {X 0,Y 374.818,Z 471.278,A -85,B 0,C 180,E1 -12328.926,E2 -12328.926} C_VEL
LIN {X 0,Y 374.847,Z 471.544,A -85,B 0,C 180,E1 -12330,E2 -12330} C_VEL
LIN {X 0,Y 374.791,Z 471.402,A -85,B 0,C 180,E1 -12331.074,E2 -12331.074} C_VEL
LIN {X 0,Y 374.788,Z 470.835,A -85,B 0,C 180,E1 -12332.149,E2 -12332.149} C_VEL
LIN {X 0,Y 374.711,Z 469.83,A -85,B 0,C 180,E1 -12333.226,E2 -12333.226} C_VEL
LIN {X 0,Y 374.647,Z 468.42,A -85,B 0,C 180,E1 -12334.303,E2 -12334.303} C_VEL
LIN {X 0,Y 374.621,Z 465.064,A -85,B 0,C 180,E1 -12336.12,E2 -12336.12} C_VEL
LIN {X 0,Y 374.765,Z 461.503,A -85,B 0,C 180,E1 -12337.543,E2 -12337.543} C_VEL
LIN {X 0,Y 374.99,Z 456.383,A -85,B 0,C 180,E1 -12339.167,E2 -12339.167} C_VEL
LIN {X 0,Y 375.425,Z 449.986,A -85,B 0,C 180,E1 -12340.79,E2 -12340.79} C_VEL
LIN {X 0,Y 376.242,Z 442.102,A -85,B 0,C 180,E1 -12342.405,E2 -12342.405} C_VEL
LIN {X 0,Y 377.014,Z 434.093,A -85,B 0,C 180,E1 -12343.75,E2 -12343.75} C_VEL
LIN {X 0,Y 378.003,Z 423.325,A -85,B 0,C 180,E1 -12345.226,E2 -12345.226} C_VEL
LIN {X 0,Y 379.216,Z 412.461,A -85,B 0,C 180,E1 -12346.417,E2 -12346.417} C_VEL
LIN {X 0,Y 380.077,Z 402.012,A -85,B 0,C 180,E1 -12347.346,E2 -12347.346} C_VEL
LIN {X 0,Y 379.441,Z 388.641,A -85,B 0,C 180,E1 -12348.353,E2 -12348.353} C_VEL
LIN {X 0,Y 378.075,Z 376.323,A -85,B 0,C 180,E1 -12349.107,E2 -12349.107} C_VEL
LIN {X 0,Y 375.465,Z 362.669,A -85,B 0,C 180,E1 -12349.789,E2 -12349.789} C_VEL
LIN {X 0,Y 375.282,Z 361.046,A -85,B 0,C 180,E1 -12349.882,E2 -12349.882} C_VEL
LIN {X 0,Y 375.726,Z 352.035,A -85,B 0,C 180,E1 -12353.573,E2 -12353.573} C_VEL
LIN {X 0,Y 376.409,Z 343.42,A -85,B 0,C 180,E1 -12357.223,E2 -12357.223} C_VEL
LIN {X 0,Y 377.214,Z 334.848,A -85,B 0,C 180,E1 -12361.014,E2 -12361.014} C_VEL
LIN {X 0,Y 378.122,Z 327.334,A -85,B 0,C 180,E1 -12364.534,E2 -12364.534} C_VEL
LIN {X 0,Y 378.553,Z 323.44,A -85,B 0,C 180,E1 -12366.448,E2 -12366.448} C_VEL
LIN {X 0,Y 378.388,Z 320.938,A -85,B 0,C 180,E1 -12367.802,E2 -12367.802} C_VEL
LIN {X 0,Y 377.547,Z 315.988,A -85,B 0,C 180,E1 -12370.657,E2 -12370.657} C_VEL
LIN {X 0,Y 376.636,Z 311.27,A -85,B 0,C 180,E1 -12373.664,E2 -12373.664} C_VEL
LIN {X 0,Y 375.938,Z 307.665,A -85,B 0,C 180,E1 -12376.235,E2 -12376.235} C_VEL
LIN {X 0,Y 375.992,Z 307.654,A -85,B 0,C 180,E1 -12380.029,E2 -12380.029} C_VEL
LIN {X 0,Y 375.967,Z 307.653,A -85,B 0,C 180,E1 -12383.496,E2 -12383.496} C_VEL
LIN {X 0,Y 375.966,Z 307.655,A -85,B 0,C 180,E1 -12385.889,E2 -12385.889} C_VEL
LIN {X 0,Y 375.969,Z 307.654,A -85,B 0,C 180,E1 -12389.688,E2 -12389.688} C_VEL
LIN {X 0,Y 376,Z 307.651,A -85,B 0,C 180,E1 -12392.141,E2 -12392.141} C_VEL
LIN {X 0,Y 376.011,Z 307.649,A -85,B 0,C 180,E1 -12394.539,E2 -12394.539} C_VEL
LIN {X 0,Y 375.968,Z 307.652,A -85,B 0,C 180,E1 -12398.046,E2 -12398.046} C_VEL
LIN {X 0,Y 376.028,Z 307.647,A -85,B 0,C 180,E1 -12401.474,E2 -12401.474} C_VEL
LIN {X 0,Y 376.063,Z 307.64,A -85,B 0,C 180,E1 -12404.833,E2 -12404.833} C_VEL
LIN {X 0,Y 376.055,Z 307.644,A -85,B 0,C 180,E1 -12408.137,E2 -12408.137} C_VEL
LIN {X 0,Y 376.197,Z 307.625,A -85,B 0,C 180,E1 -12411.947,E2 -12411.947} C_VEL
LIN {X 0,Y 376.163,Z 307.63,A -85,B 0,C 180,E1 -12414.64,E2 -12414.64} C_VEL
LIN {X 0,Y 376.356,Z 307.606,A -85,B 0,C 180,E1 -12417.859,E2 -12417.859} C_VEL
LIN {X 0,Y 376.492,Z 307.591,A -85,B 0,C 180,E1 -12420,E2 -12420} C_VEL
LIN {X 0,Y 376.193,Z 307.626,A -85,B 0,C 180,E1 -12423.213,E2 -12423.213} C_VEL
LIN {X 0,Y 376.214,Z 307.624,A -85,B 0,C 180,E1 -12426.488,E2 -12426.488} C_VEL
LIN {X 0,Y 376.077,Z 307.643,A -85,B 0,C 180,E1 -12428.598,E2 -12428.598} C_VEL
LIN {X 0,Y 375.946,Z 307.661,A -85,B 0,C 180,E1 -12429.686,E2 -12429.686} C_VEL
LIN {X 0,Y 375.868,Z 309.051,A -85,B 0,C 180,E1 -12431.869,E2 -12431.869} C_VEL
LIN {X 0,Y 375.722,Z 311.719,A -85,B 0,C 180,E1 -12435.181,E2 -12435.181} C_VEL
LIN {X 0,Y 375.574,Z 314.325,A -85,B 0,C 180,E1 -12438.302,E2 -12438.302} C_VEL
LIN {X 0,Y 380.171,Z 328.381,A -85,B 0,C 180,E1 -12439.226,E2 -12439.226} C_VEL
LIN {X 0,Y 382.547,Z 337.493,A -85,B 0,C 180,E1 -12439.925,E2 -12439.925} C_VEL
LIN {X 0,Y 382.102,Z 346.952,A -85,B 0,C 180,E1 -12440.595,E2 -12440.595} C_VEL
LIN {X 0,Y 381.144,Z 358.822,A -85,B 0,C 180,E1 -12441.641,E2 -12441.641} C_VEL
LIN {X 0,Y 380.054,Z 369.669,A -85,B 0,C 180,E1 -12442.851,E2 -12442.851} C_VEL
LIN {X 0,Y 378.95,Z 380.191,A -85,B 0,C 180,E1 -12444.333,E2 -12444.333} C_VEL
LIN {X 0,Y 378.093,Z 387.546,A -85,B 0,C 180,E1 -12445.605,E2 -12445.605} C_VEL
LIN {X 0,Y 377.273,Z 394.948,A -85,B 0,C 180,E1 -12447.165,E2 -12447.165} C_VEL
LIN {X 0,Y 376.391,Z 401.938,A -85,B 0,C 180,E1 -12449.043,E2 -12449.043} C_VEL
LIN {X 0,Y 375.854,Z 406.615,A -85,B 0,C 180,E1 -12450.667,E2 -12450.667} C_VEL
LIN {X 0,Y 375.359,Z 410.748,A -85,B 0,C 180,E1 -12452.588,E2 -12452.588} C_VEL
LIN {X 0,Y 375.004,Z 413.385,A -85,B 0,C 180,E1 -12454.45,E2 -12454.45} C_VEL
LIN {X 0,Y 374.769,Z 414.76,A -85,B 0,C 180,E1 -12456.256,E2 -12456.256} C_VEL
LIN {X 0,Y 374.693,Z 414.968,A -85,B 0,C 180,E1 -12458.241,E2 -12458.241} C_VEL
LIN {X 0,Y 374.725,Z 414.235,A -85,B 0,C 180,E1 -12459.739,E2 -12459.739} C_VEL
LIN {X 0,Y 374.881,Z 412.475,A -85,B 0,C 180,E1 -12461.418,E2 -12461.418} C_VEL
LIN {X 0,Y 375.173,Z 409.754,A -85,B 0,C 180,E1 -12463.065,E2 -12463.065} C_VEL
LIN {X 0,Y 375.445,Z 406.133,A -85,B 0,C 180,E1 -12464.657,E2 -12464.657} C_VEL
LIN {X 0,Y 375.901,Z 400.668,A -85,B 0,C 180,E1 -12466.469,E2 -12466.469} C_VEL
LIN {X 0,Y 376.463,Z 393.511,A -85,B 0,C 180,E1 -12468.309,E2 -12468.309} C_VEL
LIN {X 0,Y 377.157,Z 386.076,A -85,B 0,C 180,E1 -12469.818,E2 -12469.818} C_VEL
LIN {X 0,Y 377.957,Z 376.777,A -85,B 0,C 180,E1 -12471.35,E2 -12471.35} C_VEL
LIN {X 0,Y 378.801,Z 367.492,A -85,B 0,C 180,E1 -12472.594,E2 -12472.594} C_VEL
LIN {X 0,Y 379.652,Z 356.615,A -85,B 0,C 180,E1 -12473.774,E2 -12473.774} C_VEL
LIN {X 0,Y 380.406,Z 345.132,A -85,B 0,C 180,E1 -12474.764,E2 -12474.764} C_VEL
LIN {X 0,Y 380.983,Z 336.4,A -85,B 0,C 180,E1 -12475.367,E2 -12475.367} C_VEL
LIN {X 0,Y 379.328,Z 327.986,A -85,B 0,C 180,E1 -12475.937,E2 -12475.937} C_VEL
LIN {X 0,Y 376.017,Z 314.922,A -85,B 0,C 180,E1 -12476.659,E2 -12476.659} C_VEL
LIN {X 0,Y 375.076,Z 311.238,A -85,B 0,C 180,E1 -12476.845,E2 -12476.845} C_VEL
LIN {X 0,Y 375.127,Z 308.439,A -85,B 0,C 180,E1 -12479.612,E2 -12479.612} C_VEL
LIN {X 0,Y 375.195,Z 307.751,A -85,B 0,C 180,E1 -12480.855,E2 -12480.855} C_VEL
LIN {X 0,Y 375.652,Z 307.692,A -85,B 0,C 180,E1 -12483.899,E2 -12483.899} C_VEL
LIN {X 0,Y 375.891,Z 307.664,A -85,B 0,C 180,E1 -12486.881,E2 -12486.881} C_VEL
LIN {X 0,Y 375.997,Z 307.647,A -85,B 0,C 180,E1 -12490.339,E2 -12490.339} C_VEL
LIN {X 0,Y 376.026,Z 307.644,A -85,B 0,C 180,E1 -12493.719,E2 -12493.719} C_VEL
LIN {X 0,Y 376.104,Z 307.638,A -85,B 0,C 180,E1 -12497.042,E2 -12497.042} C_VEL
LIN {X 0,Y 376.119,Z 307.633,A -85,B 0,C 180,E1 -12500.318,E2 -12500.318} C_VEL
LIN {X 0,Y 376.214,Z 307.621,A -85,B 0,C 180,E1 -12503.564,E2 -12503.564} C_VEL
LIN {X 0,Y 376.352,Z 307.603,A -85,B 0,C 180,E1 -12507.86,E2 -12507.86} C_VEL
LIN {X 0,Y 376.488,Z 307.586,A -85,B 0,C 180,E1 -12510,E2 -12510} C_VEL
LIN {X 0,Y 376.19,Z 307.625,A -85,B 0,C 180,E1 -12513.213,E2 -12513.213} C_VEL
LIN {X 0,Y 376.214,Z 307.624,A -85,B 0,C 180,E1 -12516.436,E2 -12516.436} C_VEL
LIN {X 0,Y 376.119,Z 307.632,A -85,B 0,C 180,E1 -12519.682,E2 -12519.682} C_VEL
LIN {X 0,Y 376.09,Z 307.636,A -85,B 0,C 180,E1 -12523.658,E2 -12523.658} C_VEL
LIN {X 0,Y 376.045,Z 307.642,A -85,B 0,C 180,E1 -12527.607,E2 -12527.607} C_VEL
LIN {X 0,Y 375.979,Z 307.651,A -85,B 0,C 180,E1 -12530.832,E2 -12530.832} C_VEL
LIN {X 0,Y 375.995,Z 307.652,A -85,B 0,C 180,E1 -12534.282,E2 -12534.282} C_VEL
LIN {X 0,Y 376.021,Z 307.646,A -85,B 0,C 180,E1 -12536.652,E2 -12536.652} C_VEL
LIN {X 0,Y 375.99,Z 307.649,A -85,B 0,C 180,E1 -12537.668,E2 -12537.668} C_VEL
LIN {X 0,Y 375.344,Z 307.735,A -85,B 0,C 180,E1 -12538.562,E2 -12538.562} C_VEL
LIN {X 0,Y 372.484,Z 308.097,A -85,B 0,C 180,E1 -12540.014,E2 -12540.014} C_VEL
LIN {X 0,Y 370.041,Z 308.399,A -85,B 0,C 180,E1 -12541.189,E2 -12541.189} C_VEL
LIN {X 0,Y 368.983,Z 308.526,A -85,B 0,C 180,E1 -12542.098,E2 -12542.098} C_VEL
LIN {X 0,Y 368.893,Z 308.534,A -85,B 0,C 180,E1 -12542.406,E2 -12542.406} C_VEL
LIN {X 0,Y 368.93,Z 308.527,A -85,B 0,C 180,E1 -12545.002,E2 -12545.002} C_VEL
LIN {X 0,Y 368.909,Z 308.531,A -85,B 0,C 180,E1 -12548.64,E2 -12548.64} C_VEL
LIN {X 0,Y 368.883,Z 308.538,A -85,B 0,C 180,E1 -12552.01,E2 -12552.01} C_VEL
LIN {X 0,Y 368.881,Z 308.534,A -85,B 0,C 180,E1 -12555.176,E2 -12555.176} C_VEL
LIN {X 0,Y 368.885,Z 308.535,A -85,B 0,C 180,E1 -12558.178,E2 -12558.178} C_VEL
LIN {X 0,Y 368.912,Z 308.533,A -85,B 0,C 180,E1 -12561.36,E2 -12561.36} C_VEL
LIN {X 0,Y 368.939,Z 308.528,A -85,B 0,C 180,E1 -12565.147,E2 -12565.147} C_VEL
LIN {X 0,Y 368.932,Z 308.529,A -85,B 0,C 180,E1 -12569.047,E2 -12569.047} C_VEL
LIN {X 0,Y 368.982,Z 308.525,A -85,B 0,C 180,E1 -12571.564,E2 -12571.564} C_VEL
LIN {X 0,Y 369.002,Z 308.519,A -85,B 0,C 180,E1 -12574.02,E2 -12574.02} C_VEL
LIN {X 0,Y 368.925,Z 308.531,A -85,B 0,C 180,E1 -12577.605,E2 -12577.605} C_VEL
LIN {X 0,Y 368.958,Z 308.528,A -85,B 0,C 180,E1 -12581.106,E2 -12581.106} C_VEL
LIN {X 0,Y 369.001,Z 308.52,A -85,B 0,C 180,E1 -12584.535,E2 -12584.535} C_VEL
LIN {X 0,Y 369.009,Z 308.518,A -85,B 0,C 180,E1 -12587.907,E2 -12587.907} C_VEL
LIN {X 0,Y 369.151,Z 308.5,A -85,B 0,C 180,E1 -12591.889,E2 -12591.889} C_VEL
LIN {X 0,Y 369.144,Z 308.502,A -85,B 0,C 180,E1 -12594.538,E2 -12594.538} C_VEL
LIN {X 0,Y 369.319,Z 308.479,A -85,B 0,C 180,E1 -12597.819,E2 -12597.819} C_VEL
LIN {X 0,Y 369.459,Z 308.462,A -85,B 0,C 180,E1 -12600,E2 -12600} C_VEL
LIN {X 0,Y 369.312,Z 308.48,A -85,B 0,C 180,E1 -12602.181,E2 -12602.181} C_VEL
LIN {X 0,Y 369.177,Z 308.501,A -85,B 0,C 180,E1 -12606.559,E2 -12606.559} C_VEL
LIN {X 0,Y 369.068,Z 308.51,A -85,B 0,C 180,E1 -12609.868,E2 -12609.868} C_VEL
LIN {X 0,Y 369.041,Z 308.513,A -85,B 0,C 180,E1 -12613.772,E2 -12613.772} C_VEL
LIN {X 0,Y 368.994,Z 308.519,A -85,B 0,C 180,E1 -12617.743,E2 -12617.743} C_VEL
LIN {X 0,Y 368.913,Z 308.529,A -85,B 0,C 180,E1 -12621.221,E2 -12621.221} C_VEL
LIN {X 0,Y 368.942,Z 308.528,A -85,B 0,C 180,E1 -12624.777,E2 -12624.777} C_VEL
LIN {X 0,Y 368.934,Z 308.531,A -85,B 0,C 180,E1 -12628.44,E2 -12628.44} C_VEL
LIN {X 0,Y 368.914,Z 308.53,A -85,B 0,C 180,E1 -12630.987,E2 -12630.987} C_VEL
LIN {X 0,Y 368.94,Z 308.527,A -85,B 0,C 180,E1 -12634.853,E2 -12634.853} C_VEL
LIN {X 0,Y 368.909,Z 308.532,A -85,B 0,C 180,E1 -12638.64,E2 -12638.64} C_VEL
LIN {X 0,Y 368.883,Z 308.538,A -85,B 0,C 180,E1 -12642.009,E2 -12642.009} C_VEL
LIN {X 0,Y 368.953,Z 308.616,A -85,B 0,C 180,E1 -12645.721,E2 -12645.721} C_VEL
LIN {X 0,Y 370.23,Z 315.527,A -85,B 0,C 180,E1 -12649.404,E2 -12649.404} C_VEL
LIN {X 0,Y 371.334,Z 322.131,A -85,B 0,C 180,E1 -12652.725,E2 -12652.725} C_VEL
LIN {X 0,Y 371.335,Z 325.833,A -85,B 0,C 180,E1 -12654.472,E2 -12654.472} C_VEL
LIN {X 0,Y 370.471,Z 333.432,A -85,B 0,C 180,E1 -12657.915,E2 -12657.915} C_VEL
LIN {X 0,Y 369.642,Z 341.862,A -85,B 0,C 180,E1 -12661.619,E2 -12661.619} C_VEL
LIN {X 0,Y 368.919,Z 350.249,A -85,B 0,C 180,E1 -12665.222,E2 -12665.222} C_VEL
LIN {X 0,Y 368.296,Z 359.794,A -85,B 0,C 180,E1 -12669.235,E2 -12669.235} C_VEL
LIN {X 0,Y 368.131,Z 363.546,A -85,B 0,C 180,E1 -12670.79,E2 -12670.79} C_VEL
LIN {X 0,Y 370.138,Z 377.657,A -85,B 0,C 180,E1 -12671.383,E2 -12671.383} C_VEL
LIN {X 0,Y 371.525,Z 390.56,A -85,B 0,C 180,E1 -12672.138,E2 -12672.138} C_VEL
LIN {X 0,Y 372.323,Z 401.988,A -85,B 0,C 180,E1 -12672.987,E2 -12672.987} C_VEL
LIN {X 0,Y 371.302,Z 414.153,A -85,B 0,C 180,E1 -12674.07,E2 -12674.07} C_VEL
LIN {X 0,Y 370.368,Z 424.289,A -85,B 0,C 180,E1 -12675.213,E2 -12675.213} C_VEL
LIN {X 0,Y 369.615,Z 433.79,A -85,B 0,C 180,E1 -12676.53,E2 -12676.53} C_VEL
LIN {X 0,Y 368.913,Z 441.944,A -85,B 0,C 180,E1 -12677.904,E2 -12677.904} C_VEL
LIN {X 0,Y 368.205,Z 449.947,A -85,B 0,C 180,E1 -12679.553,E2 -12679.553} C_VEL
LIN {X 0,Y 367.864,Z 456.349,A -85,B 0,C 180,E1 -12681.208,E2 -12681.208} C_VEL
LIN {X 0,Y 367.674,Z 461.425,A -85,B 0,C 180,E1 -12682.863,E2 -12682.863} C_VEL
LIN {X 0,Y 367.624,Z 465.335,A -85,B 0,C 180,E1 -12684.515,E2 -12684.515} C_VEL
LIN {X 0,Y 367.58,Z 467.329,A -85,B 0,C 180,E1 -12685.614,E2 -12685.614} C_VEL
LIN {X 0,Y 367.634,Z 468.9,A -85,B 0,C 180,E1 -12686.712,E2 -12686.712} C_VEL
LIN {X 0,Y 367.732,Z 470.039,A -85,B 0,C 180,E1 -12687.809,E2 -12687.809} C_VEL
LIN {X 0,Y 367.743,Z 470.718,A -85,B 0,C 180,E1 -12688.905,E2 -12688.905} C_VEL
LIN {X 0,Y 367.768,Z 470.995,A -85,B 0,C 180,E1 -12690,E2 -12690} C_VEL
LIN {X 0,Y 367.717,Z 470.865,A -85,B 0,C 180,E1 -12691.095,E2 -12691.095} C_VEL
LIN {X 0,Y 367.72,Z 470.321,A -85,B 0,C 180,E1 -12692.191,E2 -12692.191} C_VEL
LIN {X 0,Y 367.614,Z 469.326,A -85,B 0,C 180,E1 -12693.288,E2 -12693.288} C_VEL
LIN {X 0,Y 367.57,Z 467.925,A -85,B 0,C 180,E1 -12694.386,E2 -12694.386} C_VEL
LIN {X 0,Y 367.525,Z 464.915,A -85,B 0,C 180,E1 -12696.08,E2 -12696.08} C_VEL
LIN {X 0,Y 367.691,Z 461.052,A -85,B 0,C 180,E1 -12697.689,E2 -12697.689} C_VEL
LIN {X 0,Y 367.942,Z 455.973,A -85,B 0,C 180,E1 -12699.344,E2 -12699.344} C_VEL
LIN {X 0,Y 368.411,Z 449.627,A -85,B 0,C 180,E1 -12700.998,E2 -12700.998} C_VEL
LIN {X 0,Y 369.276,Z 441.804,A -85,B 0,C 180,E1 -12702.643,E2 -12702.643} C_VEL
LIN {X 0,Y 370.094,Z 433.854,A -85,B 0,C 180,E1 -12704.012,E2 -12704.012} C_VEL
LIN {X 0,Y 371.014,Z 424.226,A -85,B 0,C 180,E1 -12705.379,E2 -12705.379} C_VEL
LIN {X 0,Y 372.251,Z 413.666,A -85,B 0,C 180,E1 -12706.592,E2 -12706.592} C_VEL
LIN {X 0,Y 373.206,Z 403.625,A -85,B 0,C 180,E1 -12707.536,E2 -12707.536} C_VEL
LIN {X 0,Y 372.84,Z 391.298,A -85,B 0,C 180,E1 -12708.537,E2 -12708.537} C_VEL
LIN {X 0,Y 371.495,Z 378.199,A -85,B 0,C 180,E1 -12709.405,E2 -12709.405} C_VEL
LIN {X 0,Y 368.999,Z 364.283,A -85,B 0,C 180,E1 -12710.158,E2 -12710.158} C_VEL
LIN {X 0,Y 368.228,Z 360.484,A -85,B 0,C 180,E1 -12710.335,E2 -12710.335} C_VEL
LIN {X 0,Y 368.712,Z 352.23,A -85,B 0,C 180,E1 -12713.804,E2 -12713.804} C_VEL
LIN {X 0,Y 369.453,Z 343.098,A -85,B 0,C 180,E1 -12717.779,E2 -12717.779} C_VEL
LIN {X 0,Y 370.249,Z 335.316,A -85,B 0,C 180,E1 -12721.33,E2 -12721.33} C_VEL
LIN {X 0,Y 371.155,Z 328.468,A -85,B 0,C 180,E1 -12724.616,E2 -12724.616} C_VEL
LIN {X 0,Y 371.607,Z 324.595,A -85,B 0,C 180,E1 -12726.566,E2 -12726.566} C_VEL
LIN {X 0,Y 371.173,Z 320.805,A -85,B 0,C 180,E1 -12728.671,E2 -12728.671} C_VEL
LIN {X 0,Y 370.332,Z 315.967,A -85,B 0,C 180,E1 -12731.623,E2 -12731.623} C_VEL
LIN {X 0,Y 369.317,Z 310.656,A -85,B 0,C 180,E1 -12735.243,E2 -12735.243} C_VEL
LIN {X 0,Y 368.904,Z 308.54,A -85,B 0,C 180,E1 -12736.873,E2 -12736.873} C_VEL
LIN {X 0,Y 368.915,Z 308.537,A -85,B 0,C 180,E1 -12739.643,E2 -12739.643} C_VEL
LIN {X 0,Y 368.905,Z 308.533,A -85,B 0,C 180,E1 -12743.144,E2 -12743.144} C_VEL
LIN {X 0,Y 368.902,Z 308.535,A -85,B 0,C 180,E1 -12746.462,E2 -12746.462} C_VEL
LIN {X 0,Y 368.933,Z 308.531,A -85,B 0,C 180,E1 -12749.047,E2 -12749.047} C_VEL
LIN {X 0,Y 368.984,Z 308.524,A -85,B 0,C 180,E1 -12751.564,E2 -12751.564} C_VEL
LIN {X 0,Y 369.004,Z 308.522,A -85,B 0,C 180,E1 -12754.02,E2 -12754.02} C_VEL
LIN {X 0,Y 368.937,Z 308.527,A -85,B 0,C 180,E1 -12757.605,E2 -12757.605} C_VEL
LIN {X 0,Y 368.987,Z 308.525,A -85,B 0,C 180,E1 -12761.107,E2 -12761.107} C_VEL
LIN {X 0,Y 369.003,Z 308.518,A -85,B 0,C 180,E1 -12764.535,E2 -12764.535} C_VEL
LIN {X 0,Y 369.01,Z 308.522,A -85,B 0,C 180,E1 -12767.907,E2 -12767.907} C_VEL
LIN {X 0,Y 369.095,Z 308.508,A -85,B 0,C 180,E1 -12771.238,E2 -12771.238} C_VEL
LIN {X 0,Y 369.135,Z 308.506,A -85,B 0,C 180,E1 -12774.537,E2 -12774.537} C_VEL
LIN {X 0,Y 369.321,Z 308.482,A -85,B 0,C 180,E1 -12777.819,E2 -12777.819} C_VEL
LIN {X 0,Y 369.462,Z 308.466,A -85,B 0,C 180,E1 -12780,E2 -12780} C_VEL
LIN {X 0,Y 369.324,Z 308.482,A -85,B 0,C 180,E1 -12782.181,E2 -12782.181} C_VEL
LIN {X 0,Y 369.179,Z 308.501,A -85,B 0,C 180,E1 -12786.559,E2 -12786.559} C_VEL
LIN {X 0,Y 369.009,Z 308.524,A -85,B 0,C 180,E1 -12788.764,E2 -12788.764} C_VEL
LIN {X 0,Y 368.89,Z 308.633,A -85,B 0,C 180,E1 -12789.873,E2 -12789.873} C_VEL
LIN {X 0,Y 368.8,Z 311.534,A -85,B 0,C 180,E1 -12793.618,E2 -12793.618} C_VEL
LIN {X 0,Y 368.601,Z 313.955,A -85,B 0,C 180,E1 -12796.619,E2 -12796.619} C_VEL
LIN {X 0,Y 368.576,Z 314.989,A -85,B 0,C 180,E1 -12797.844,E2 -12797.844} C_VEL
LIN {X 0,Y 373.038,Z 328.25,A -85,B 0,C 180,E1 -12798.737,E2 -12798.737} C_VEL
LIN {X 0,Y 375.748,Z 338.332,A -85,B 0,C 180,E1 -12799.532,E2 -12799.532} C_VEL
LIN {X 0,Y 376.009,Z 341.057,A -85,B 0,C 180,E1 -12799.738,E2 -12799.738} C_VEL
LIN {X 0,Y 375.013,Z 353.226,A -85,B 0,C 180,E1 -12800.693,E2 -12800.693} C_VEL
LIN {X 0,Y 373.96,Z 364.168,A -85,B 0,C 180,E1 -12801.788,E2 -12801.788} C_VEL
LIN {X 0,Y 372.999,Z 373.408,A -85,B 0,C 180,E1 -12802.933,E2 -12802.933} C_VEL
LIN {X 0,Y 371.968,Z 382.239,A -85,B 0,C 180,E1 -12804.264,E2 -12804.264} C_VEL
LIN {X 0,Y 370.962,Z 390.662,A -85,B 0,C 180,E1 -12805.832,E2 -12805.832} C_VEL
LIN {X 0,Y 370.102,Z 397.555,A -85,B 0,C 180,E1 -12807.419,E2 -12807.419} C_VEL
LIN {X 0,Y 369.279,Z 403.862,A -85,B 0,C 180,E1 -12809.25,E2 -12809.25} C_VEL
LIN {X 0,Y 368.723,Z 408.382,A -85,B 0,C 180,E1 -12810.973,E2 -12810.973} C_VEL
LIN {X 0,Y 368.243,Z 412.033,A -85,B 0,C 180,E1 -12812.885,E2 -12812.885} C_VEL
LIN {X 0,Y 367.862,Z 414.549,A -85,B 0,C 180,E1 -12814.97,E2 -12814.97} C_VEL
LIN {X 0,Y 367.67,Z 415.467,A -85,B 0,C 180,E1 -12816.598,E2 -12816.598} C_VEL
LIN {X 0,Y 367.614,Z 415.472,A -85,B 0,C 180,E1 -12818.387,E2 -12818.387} C_VEL
LIN {X 0,Y 367.688,Z 414.073,A -85,B 0,C 180,E1 -12820.532,E2 -12820.532} C_VEL
LIN {X 0,Y 368.024,Z 411.086,A -85,B 0,C 180,E1 -12822.682,E2 -12822.682} C_VEL
LIN {X 0,Y 368.279,Z 408.073,A -85,B 0,C 180,E1 -12824.152,E2 -12824.152} C_VEL
LIN {X 0,Y 368.714,Z 402.929,A -85,B 0,C 180,E1 -12826.052,E2 -12826.052} C_VEL
LIN {X 0,Y 369.153,Z 397.549,A -85,B 0,C 180,E1 -12827.595,E2 -12827.595} C_VEL
LIN {X 0,Y 369.778,Z 390.951,A -85,B 0,C 180,E1 -12829.131,E2 -12829.131} C_VEL
LIN {X 0,Y 370.547,Z 382.234,A -85,B 0,C 180,E1 -12830.766,E2 -12830.766} C_VEL
LIN {X 0,Y 371.419,Z 373.128,A -85,B 0,C 180,E1 -12832.15,E2 -12832.15} C_VEL
LIN {X 0,Y 372.257,Z 363.588,A -85,B 0,C 180,E1 -12833.339,E2 -12833.339} C_VEL
LIN {X 0,Y 373.039,Z 352.818,A -85,B 0,C 180,E1 -12834.431,E2 -12834.431} C_VEL
LIN {X 0,Y 373.896,Z 341.297,A -85,B 0,C 180,E1 -12835.347,E2 -12835.347} C_VEL
LIN {X 0,Y 374.039,Z 336.268,A -85,B 0,C 180,E1 -12835.689,E2 -12835.689} C_VEL
LIN {X 0,Y 371.071,Z 323.334,A -85,B 0,C 180,E1 -12836.55,E2 -12836.55} C_VEL
LIN {X 0,Y 368.034,Z 311.719,A -85,B 0,C 180,E1 -12837.164,E2 -12837.164} C_VEL
LIN {X 0,Y 368.077,Z 308.647,A -85,B 0,C 180,E1 -12840.235,E2 -12840.235} C_VEL
LIN {X 0,Y 368.613,Z 308.568,A -85,B 0,C 180,E1 -12843.99,E2 -12843.99} C_VEL
LIN {X 0,Y 368.846,Z 308.538,A -85,B 0,C 180,E1 -12846.413,E2 -12846.413} C_VEL
LIN {X 0,Y 368.93,Z 308.527,A -85,B 0,C 180,E1 -12849.946,E2 -12849.946} C_VEL
LIN {X 0,Y 368.969,Z 308.525,A -85,B 0,C 180,E1 -12853.398,E2 -12853.398} C_VEL
LIN {X 0,Y 369.059,Z 308.515,A -85,B 0,C 180,E1 -12856.79,E2 -12856.79} C_VEL
LIN {X 0,Y 369.068,Z 308.511,A -85,B 0,C 180,E1 -12860.132,E2 -12860.132} C_VEL
LIN {X 0,Y 369.174,Z 308.499,A -85,B 0,C 180,E1 -12863.441,E2 -12863.441} C_VEL
LIN {X 0,Y 369.317,Z 308.479,A -85,B 0,C 180,E1 -12867.819,E2 -12867.819} C_VEL
LIN {X 0,Y 369.458,Z 308.462,A -85,B 0,C 180,E1 -12870,E2 -12870} C_VEL
LIN {X 0,Y 369.32,Z 308.481,A -85,B 0,C 180,E1 -12872.181,E2 -12872.181} C_VEL
LIN {X 0,Y 369.174,Z 308.501,A -85,B 0,C 180,E1 -12876.559,E2 -12876.559} C_VEL
LIN {X 0,Y 369.068,Z 308.511,A -85,B 0,C 180,E1 -12879.868,E2 -12879.868} C_VEL
LIN {X 0,Y 369.038,Z 308.515,A -85,B 0,C 180,E1 -12883.772,E2 -12883.772} C_VEL
LIN {X 0,Y 369.002,Z 308.52,A -85,B 0,C 180,E1 -12887.768,E2 -12887.768} C_VEL
LIN {X 0,Y 368.93,Z 308.528,A -85,B 0,C 180,E1 -12891.22,E2 -12891.22} C_VEL
LIN {X 0,Y 368.959,Z 308.525,A -85,B 0,C 180,E1 -12894.775,E2 -12894.775} C_VEL
LIN {X 0,Y 368.954,Z 308.523,A -85,B 0,C 180,E1 -12897.667,E2 -12897.667} C_VEL
LIN {X 0,Y 368.911,Z 308.53,A -85,B 0,C 180,E1 -12900.988,E2 -12900.988} C_VEL
LIN {X 0,Y 368.893,Z 308.534,A -85,B 0,C 180,E1 -12902.406,E2 -12902.406} C_VEL
LIN {X 0,Y 368.226,Z 308.617,A -85,B 0,C 180,E1 -12903.317,E2 -12903.317} C_VEL
LIN {X 0,Y 365.407,Z 308.968,A -85,B 0,C 180,E1 -12904.801,E2 -12904.801} C_VEL
LIN {X 0,Y 363.011,Z 309.27,A -85,B 0,C 180,E1 -12906.001,E2 -12906.001} C_VEL
LIN {X 0,Y 361.961,Z 309.398,A -85,B 0,C 180,E1 -12906.928,E2 -12906.928} C_VEL
LIN {X 0,Y 361.864,Z 309.408,A -85,B 0,C 180,E1 -12907.242,E2 -12907.242} C_VEL
LIN {X 0,Y 361.837,Z 309.411,A -85,B 0,C 180,E1 -12910.756,E2 -12910.756} C_VEL
LIN {X 0,Y 361.819,Z 309.414,A -85,B 0,C 180,E1 -12914.369,E2 -12914.369} C_VEL
LIN {X 0,Y 361.838,Z 309.414,A -85,B 0,C 180,E1 -12917.568,E2 -12917.568} C_VEL
LIN {X 0,Y 361.872,Z 309.407,A -85,B 0,C 180,E1 -12920.973,E2 -12920.973} C_VEL
LIN {X 0,Y 361.876,Z 309.406,A -85,B 0,C 180,E1 -12924.655,E2 -12924.655} C_VEL
LIN {X 0,Y 361.84,Z 309.411,A -85,B 0,C 180,E1 -12928.371,E2 -12928.371} C_VEL
LIN {X 0,Y 361.903,Z 309.404,A -85,B 0,C 180,E1 -12930.956,E2 -12930.956} C_VEL
LIN {X 0,Y 361.957,Z 309.401,A -85,B 0,C 180,E1 -12933.475,E2 -12933.475} C_VEL
LIN {X 0,Y 361.882,Z 309.409,A -85,B 0,C 180,E1 -12937.144,E2 -12937.144} C_VEL
LIN {X 0,Y 361.889,Z 309.406,A -85,B 0,C 180,E1 -12940.723,E2 -12940.723} C_VEL
LIN {X 0,Y 361.947,Z 309.397,A -85,B 0,C 180,E1 -12944.226,E2 -12944.226} C_VEL
LIN {X 0,Y 362.003,Z 309.391,A -85,B 0,C 180,E1 -12946.528,E2 -12946.528} C_VEL
LIN {X 0,Y 362.004,Z 309.39,A -85,B 0,C 180,E1 -12949.937,E2 -12949.937} C_VEL
LIN {X 0,Y 362.156,Z 309.374,A -85,B 0,C 180,E1 -12953.314,E2 -12953.314} C_VEL
LIN {X 0,Y 362.282,Z 309.355,A -85,B 0,C 180,E1 -12957.777,E2 -12957.777} C_VEL
LIN {X 0,Y 362.429,Z 309.337,A -85,B 0,C 180,E1 -12960,E2 -12960} C_VEL
LIN {X 0,Y 362.275,Z 309.357,A -85,B 0,C 180,E1 -12962.224,E2 -12962.224} C_VEL
LIN {X 0,Y 362.139,Z 309.378,A -85,B 0,C 180,E1 -12966.687,E2 -12966.687} C_VEL
LIN {X 0,Y 362.004,Z 309.391,A -85,B 0,C 180,E1 -12970.063,E2 -12970.063} C_VEL
LIN {X 0,Y 362.002,Z 309.39,A -85,B 0,C 180,E1 -12973.899,E2 -12973.899} C_VEL
LIN {X 0,Y 361.932,Z 309.401,A -85,B 0,C 180,E1 -12976.934,E2 -12976.934} C_VEL
LIN {X 0,Y 361.89,Z 309.409,A -85,B 0,C 180,E1 -12980.461,E2 -12980.461} C_VEL
LIN {X 0,Y 361.897,Z 309.407,A -85,B 0,C 180,E1 -12984.113,E2 -12984.113} C_VEL
LIN {X 0,Y 361.868,Z 309.409,A -85,B 0,C 180,E1 -12987.783,E2 -12987.783} C_VEL
LIN {X 0,Y 361.85,Z 309.409,A -85,B 0,C 180,E1 -12991.285,E2 -12991.285} C_VEL
LIN {X 0,Y 361.858,Z 309.412,A -85,B 0,C 180,E1 -12994.28,E2 -12994.28} C_VEL
LIN {X 0,Y 361.866,Z 309.407,A -85,B 0,C 180,E1 -12997.223,E2 -12997.223} C_VEL
LIN {X 0,Y 361.837,Z 309.415,A -85,B 0,C 180,E1 -13000.755,E2 -13000.755} C_VEL
LIN {X 0,Y 361.82,Z 309.416,A -85,B 0,C 180,E1 -13004.368,E2 -13004.368} C_VEL
LIN {X 0,Y 361.899,Z 309.541,A -85,B 0,C 180,E1 -13005.441,E2 -13005.441} C_VEL
LIN {X 0,Y 363.08,Z 316.1,A -85,B 0,C 180,E1 -13009.018,E2 -13009.018} C_VEL
LIN {X 0,Y 364.213,Z 322.43,A -85,B 0,C 180,E1 -13012.294,E2 -13012.294} C_VEL
LIN {X 0,Y 364.37,Z 326.149,A -85,B 0,C 180,E1 -13014.106,E2 -13014.106} C_VEL
LIN {X 0,Y 363.57,Z 332.872,A -85,B 0,C 180,E1 -13017.231,E2 -13017.231} C_VEL
LIN {X 0,Y 362.713,Z 341.285,A -85,B 0,C 180,E1 -13021.026,E2 -13021.026} C_VEL
LIN {X 0,Y 361.928,Z 349.674,A -85,B 0,C 180,E1 -13024.71,E2 -13024.71} C_VEL
LIN {X 0,Y 361.317,Z 357.995,A -85,B 0,C 180,E1 -13028.311,E2 -13028.311} C_VEL
LIN {X 0,Y 361.082,Z 363.029,A -85,B 0,C 180,E1 -13030.456,E2 -13030.456} C_VEL
LIN {X 0,Y 363.15,Z 377.907,A -85,B 0,C 180,E1 -13031.107,E2 -13031.107} C_VEL
LIN {X 0,Y 364.606,Z 391.49,A -85,B 0,C 180,E1 -13031.937,E2 -13031.937} C_VEL
LIN {X 0,Y 365.352,Z 402.547,A -85,B 0,C 180,E1 -13032.797,E2 -13032.797} C_VEL
LIN {X 0,Y 364.305,Z 414.437,A -85,B 0,C 180,E1 -13033.9,E2 -13033.9} C_VEL
LIN {X 0,Y 363.291,Z 425.071,A -85,B 0,C 180,E1 -13035.148,E2 -13035.148} C_VEL
LIN {X 0,Y 362.483,Z 434.712,A -85,B 0,C 180,E1 -13036.546,E2 -13036.546} C_VEL
LIN {X 0,Y 361.772,Z 442.627,A -85,B 0,C 180,E1 -13037.946,E2 -13037.946} C_VEL
LIN {X 0,Y 361.1,Z 450.353,A -85,B 0,C 180,E1 -13039.628,E2 -13039.628} C_VEL
LIN {X 0,Y 360.733,Z 457.482,A -85,B 0,C 180,E1 -13041.598,E2 -13041.598} C_VEL
LIN {X 0,Y 360.569,Z 462.199,A -85,B 0,C 180,E1 -13043.284,E2 -13043.284} C_VEL
LIN {X 0,Y 360.51,Z 465.77,A -85,B 0,C 180,E1 -13044.967,E2 -13044.967} C_VEL
LIN {X 0,Y 360.543,Z 468.298,A -85,B 0,C 180,E1 -13046.648,E2 -13046.648} C_VEL
LIN {X 0,Y 360.664,Z 469.463,A -85,B 0,C 180,E1 -13047.766,E2 -13047.766} C_VEL
LIN {X 0,Y 360.67,Z 470.158,A -85,B 0,C 180,E1 -13048.883,E2 -13048.883} C_VEL
LIN {X 0,Y 360.691,Z 470.446,A -85,B 0,C 180,E1 -13050,E2 -13050} C_VEL
LIN {X 0,Y 360.646,Z 470.328,A -85,B 0,C 180,E1 -13051.117,E2 -13051.117} C_VEL
LIN {X 0,Y 360.652,Z 469.806,A -85,B 0,C 180,E1 -13052.234,E2 -13052.234} C_VEL
LIN {X 0,Y 360.494,Z 467.438,A -85,B 0,C 180,E1 -13054.473,E2 -13054.473} C_VEL
LIN {X 0,Y 360.429,Z 464.788,A -85,B 0,C 180,E1 -13056.038,E2 -13056.038} C_VEL
LIN {X 0,Y 360.618,Z 460.633,A -85,B 0,C 180,E1 -13057.841,E2 -13057.841} C_VEL
LIN {X 0,Y 360.908,Z 455.586,A -85,B 0,C 180,E1 -13059.528,E2 -13059.528} C_VEL
LIN {X 0,Y 361.396,Z 449.272,A -85,B 0,C 180,E1 -13061.214,E2 -13061.214} C_VEL
LIN {X 0,Y 362.313,Z 441.495,A -85,B 0,C 180,E1 -13062.89,E2 -13062.89} C_VEL
LIN {X 0,Y 363.179,Z 433.603,A -85,B 0,C 180,E1 -13064.284,E2 -13064.284} C_VEL
LIN {X 0,Y 364.142,Z 424.072,A -85,B 0,C 180,E1 -13065.676,E2 -13065.676} C_VEL
LIN {X 0,Y 365.456,Z 413.64,A -85,B 0,C 180,E1 -13066.91,E2 -13066.91} C_VEL
LIN {X 0,Y 366.393,Z 403.768,A -85,B 0,C 180,E1 -13067.873,E2 -13067.873} C_VEL
LIN {X 0,Y 366.059,Z 391.769,A -85,B 0,C 180,E1 -13068.888,E2 -13068.888} C_VEL
LIN {X 0,Y 365.001,Z 380.377,A -85,B 0,C 180,E1 -13069.691,E2 -13069.691} C_VEL
LIN {X 0,Y 362.67,Z 366.787,A -85,B 0,C 180,E1 -13070.485,E2 -13070.485} C_VEL
LIN {X 0,Y 361.229,Z 359.868,A -85,B 0,C 180,E1 -13070.829,E2 -13070.829} C_VEL
LIN {X 0,Y 361.79,Z 350.954,A -85,B 0,C 180,E1 -13074.687,E2 -13074.687} C_VEL
LIN {X 0,Y 362.532,Z 342.785,A -85,B 0,C 180,E1 -13078.357,E2 -13078.357} C_VEL
LIN {X 0,Y 363.641,Z 333.452,A -85,B 0,C 180,E1 -13082.762,E2 -13082.762} C_VEL
LIN {X 0,Y 364.529,Z 327.164,A -85,B 0,C 180,E1 -13085.929,E2 -13085.929} C_VEL
LIN {X 0,Y 364.471,Z 323.8,A -85,B 0,C 180,E1 -13087.759,E2 -13087.759} C_VEL
LIN {X 0,Y 363.561,Z 318.33,A -85,B 0,C 180,E1 -13091.091,E2 -13091.091} C_VEL
LIN {X 0,Y 362.683,Z 313.694,A -85,B 0,C 180,E1 -13094.235,E2 -13094.235} C_VEL
LIN {X 0,Y 361.86,Z 309.419,A -85,B 0,C 180,E1 -13097.564,E2 -13097.564} C_VEL
LIN {X 0,Y 361.874,Z 309.411,A -85,B 0,C 180,E1 -13101.576,E2 -13101.576} C_VEL
LIN {X 0,Y 361.878,Z 309.41,A -85,B 0,C 180,E1 -13104.655,E2 -13104.655} C_VEL
LIN {X 0,Y 361.842,Z 309.414,A -85,B 0,C 180,E1 -13108.371,E2 -13108.371} C_VEL
LIN {X 0,Y 361.904,Z 309.406,A -85,B 0,C 180,E1 -13110.955,E2 -13110.955} C_VEL
LIN {X 0,Y 361.959,Z 309.399,A -85,B 0,C 180,E1 -13113.475,E2 -13113.475} C_VEL
LIN {X 0,Y 361.895,Z 309.406,A -85,B 0,C 180,E1 -13117.145,E2 -13117.145} C_VEL
LIN {X 0,Y 361.925,Z 309.403,A -85,B 0,C 180,E1 -13120.724,E2 -13120.724} C_VEL
LIN {X 0,Y 361.951,Z 309.397,A -85,B 0,C 180,E1 -13124.226,E2 -13124.226} C_VEL
LIN {X 0,Y 362.003,Z 309.391,A -85,B 0,C 180,E1 -13126.528,E2 -13126.528} C_VEL
LIN {X 0,Y 362.005,Z 309.394,A -85,B 0,C 180,E1 -13129.937,E2 -13129.937} C_VEL
LIN {X 0,Y 362.139,Z 309.374,A -85,B 0,C 180,E1 -13133.313,E2 -13133.313} C_VEL
LIN {X 0,Y 362.285,Z 309.358,A -85,B 0,C 180,E1 -13137.776,E2 -13137.776} C_VEL
LIN {X 0,Y 362.431,Z 309.342,A -85,B 0,C 180,E1 -13140,E2 -13140} C_VEL
LIN {X 0,Y 362.288,Z 309.358,A -85,B 0,C 180,E1 -13142.223,E2 -13142.223} C_VEL
LIN {X 0,Y 362.141,Z 309.377,A -85,B 0,C 180,E1 -13146.687,E2 -13146.687} C_VEL
LIN {X 0,Y 361.943,Z 309.404,A -85,B 0,C 180,E1 -13148.936,E2 -13148.936} C_VEL
LIN {X 0,Y 361.88,Z 310.775,A -85,B 0,C 180,E1 -13151.198,E2 -13151.198} C_VEL
LIN {X 0,Y 361.79,Z 312.734,A -85,B 0,C 180,E1 -13153.762,E2 -13153.762} C_VEL
LIN {X 0,Y 361.552,Z 315.607,A -85,B 0,C 180,E1 -13157.335,E2 -13157.335} C_VEL
LIN {X 0,Y 366.117,Z 328.804,A -85,B 0,C 180,E1 -13158.277,E2 -13158.277} C_VEL
LIN {X 0,Y 369.353,Z 340.968,A -85,B 0,C 180,E1 -13159.277,E2 -13159.277} C_VEL
LIN {X 0,Y 368.474,Z 353.204,A -85,B 0,C 180,E1 -13160.25,E2 -13160.25} C_VEL
LIN {X 0,Y 367.251,Z 365.208,A -85,B 0,C 180,E1 -13161.468,E2 -13161.468} C_VEL
LIN {X 0,Y 366.057,Z 375.802,A -85,B 0,C 180,E1 -13162.843,E2 -13162.843} C_VEL
LIN {X 0,Y 365.011,Z 384.026,A -85,B 0,C 180,E1 -13164.151,E2 -13164.151} C_VEL
LIN {X 0,Y 363.997,Z 392.212,A -85,B 0,C 180,E1 -13165.749,E2 -13165.749} C_VEL
LIN {X 0,Y 363.092,Z 398.877,A -85,B 0,C 180,E1 -13167.354,E2 -13167.354} C_VEL
LIN {X 0,Y 362.253,Z 404.879,A -85,B 0,C 180,E1 -13169.186,E2 -13169.186} C_VEL
LIN {X 0,Y 361.626,Z 409.894,A -85,B 0,C 180,E1 -13171.227,E2 -13171.227} C_VEL
LIN {X 0,Y 361.12,Z 413.287,A -85,B 0,C 180,E1 -13173.19,E2 -13173.19} C_VEL
LIN {X 0,Y 360.768,Z 415.293,A -85,B 0,C 180,E1 -13175.096,E2 -13175.096} C_VEL
LIN {X 0,Y 360.559,Z 416.134,A -85,B 0,C 180,E1 -13177.175,E2 -13177.175} C_VEL
LIN {X 0,Y 360.547,Z 415.862,A -85,B 0,C 180,E1 -13178.766,E2 -13178.766} C_VEL
LIN {X 0,Y 360.622,Z 414.605,A -85,B 0,C 180,E1 -13180.53,E2 -13180.53} C_VEL
LIN {X 0,Y 360.87,Z 412.373,A -85,B 0,C 180,E1 -13182.263,E2 -13182.263} C_VEL
LIN {X 0,Y 361.162,Z 409.218,A -85,B 0,C 180,E1 -13183.945,E2 -13183.945} C_VEL
LIN {X 0,Y 361.613,Z 403.959,A -85,B 0,C 180,E1 -13185.98,E2 -13185.98} C_VEL
LIN {X 0,Y 362.173,Z 397.644,A -85,B 0,C 180,E1 -13187.837,E2 -13187.837} C_VEL
LIN {X 0,Y 362.819,Z 390.932,A -85,B 0,C 180,E1 -13189.401,E2 -13189.401} C_VEL
LIN {X 0,Y 363.665,Z 381.936,A -85,B 0,C 180,E1 -13191.091,E2 -13191.091} C_VEL
LIN {X 0,Y 364.662,Z 371.79,A -85,B 0,C 180,E1 -13192.62,E2 -13192.62} C_VEL
LIN {X 0,Y 365.638,Z 360.794,A -85,B 0,C 180,E1 -13193.938,E2 -13193.938} C_VEL
LIN {X 0,Y 366.45,Z 349.675,A -85,B 0,C 180,E1 -13195.009,E2 -13195.009} C_VEL
LIN {X 0,Y 367.257,Z 338.001,A -85,B 0,C 180,E1 -13195.886,E2 -13195.886} C_VEL
LIN {X 0,Y 364.307,Z 324.969,A -85,B 0,C 180,E1 -13196.785,E2 -13196.785} C_VEL
LIN {X 0,Y 360.972,Z 312.199,A -85,B 0,C 180,E1 -13197.483,E2 -13197.483} C_VEL
LIN {X 0,Y 361.006,Z 310.098,A -85,B 0,C 180,E1 -13199.591,E2 -13199.591} C_VEL
LIN {X 0,Y 361.154,Z 309.501,A -85,B 0,C 180,E1 -13201.127,E2 -13201.127} C_VEL
LIN {X 0,Y 361.485,Z 309.459,A -85,B 0,C 180,E1 -13203.438,E2 -13203.438} C_VEL
LIN {X 0,Y 361.731,Z 309.425,A -85,B 0,C 180,E1 -13205.945,E2 -13205.945} C_VEL
LIN {X 0,Y 361.883,Z 309.407,A -85,B 0,C 180,E1 -13209.539,E2 -13209.539} C_VEL
LIN {X 0,Y 361.929,Z 309.404,A -85,B 0,C 180,E1 -13213.066,E2 -13213.066} C_VEL
LIN {X 0,Y 362,Z 309.392,A -85,B 0,C 180,E1 -13216.528,E2 -13216.528} C_VEL
LIN {X 0,Y 362.032,Z 309.387,A -85,B 0,C 180,E1 -13219.938,E2 -13219.938} C_VEL
LIN {X 0,Y 362.136,Z 309.376,A -85,B 0,C 180,E1 -13223.313,E2 -13223.313} C_VEL
LIN {X 0,Y 362.281,Z 309.356,A -85,B 0,C 180,E1 -13227.776,E2 -13227.776} C_VEL
LIN {X 0,Y 362.427,Z 309.337,A -85,B 0,C 180,E1 -13230,E2 -13230} C_VEL
LIN {X 0,Y 362.284,Z 309.357,A -85,B 0,C 180,E1 -13232.224,E2 -13232.224} C_VEL
LIN {X 0,Y 362.136,Z 309.378,A -85,B 0,C 180,E1 -13236.687,E2 -13236.687} C_VEL
LIN {X 0,Y 362.032,Z 309.388,A -85,B 0,C 180,E1 -13240.062,E2 -13240.062} C_VEL
LIN {X 0,Y 361.999,Z 309.392,A -85,B 0,C 180,E1 -13243.899,E2 -13243.899} C_VEL
LIN {X 0,Y 361.968,Z 309.397,A -85,B 0,C 180,E1 -13247.939,E2 -13247.939} C_VEL
LIN {X 0,Y 361.893,Z 309.405,A -85,B 0,C 180,E1 -13251.653,E2 -13251.653} C_VEL
LIN {X 0,Y 361.93,Z 309.399,A -85,B 0,C 180,E1 -13255.29,E2 -13255.29} C_VEL
LIN {X 0,Y 361.92,Z 309.403,A -85,B 0,C 180,E1 -13257.778,E2 -13257.778} C_VEL
LIN {X 0,Y 361.848,Z 309.41,A -85,B 0,C 180,E1 -13261.285,E2 -13261.285} C_VEL
LIN {X 0,Y 361.855,Z 309.412,A -85,B 0,C 180,E1 -13264.281,E2 -13264.281} C_VEL
LIN {X 0,Y 361.864,Z 309.408,A -85,B 0,C 180,E1 -13267.242,E2 -13267.242} C_VEL
LIN {X 0,Y 361.155,Z 309.5,A -85,B 0,C 180,E1 -13268.171,E2 -13268.171} C_VEL
LIN {X 0,Y 358.263,Z 309.859,A -85,B 0,C 180,E1 -13269.679,E2 -13269.679} C_VEL
LIN {X 0,Y 355.855,Z 310.156,A -85,B 0,C 180,E1 -13270.9,E2 -13270.9} C_VEL
LIN {X 0,Y 354.852,Z 310.286,A -85,B 0,C 180,E1 -13271.845,E2 -13271.845} C_VEL
LIN {X 0,Y 354.786,Z 310.289,A -85,B 0,C 180,E1 -13272.165,E2 -13272.165} C_VEL
LIN {X 0,Y 354.769,Z 310.294,A -85,B 0,C 180,E1 -13276.104,E2 -13276.104} C_VEL
LIN {X 0,Y 354.79,Z 310.29,A -85,B 0,C 180,E1 -13279.179,E2 -13279.179} C_VEL
LIN {X 0,Y 354.81,Z 310.286,A -85,B 0,C 180,E1 -13282.403,E2 -13282.403} C_VEL
LIN {X 0,Y 354.814,Z 310.286,A -85,B 0,C 180,E1 -13284.941,E2 -13284.941} C_VEL
LIN {X 0,Y 354.795,Z 310.288,A -85,B 0,C 180,E1 -13288.405,E2 -13288.405} C_VEL
LIN {X 0,Y 354.854,Z 310.285,A -85,B 0,C 180,E1 -13291.619,E2 -13291.619} C_VEL
LIN {X 0,Y 354.901,Z 310.275,A -85,B 0,C 180,E1 -13294.173,E2 -13294.173} C_VEL
LIN {X 0,Y 354.819,Z 310.286,A -85,B 0,C 180,E1 -13297.893,E2 -13297.893} C_VEL
LIN {X 0,Y 354.893,Z 310.276,A -85,B 0,C 180,E1 -13301.908,E2 -13301.908} C_VEL
LIN {X 0,Y 354.946,Z 310.269,A -85,B 0,C 180,E1 -13305.981,E2 -13305.981} C_VEL
LIN {X 0,Y 354.96,Z 310.268,A -85,B 0,C 180,E1 -13309.736,E2 -13309.736} C_VEL
LIN {X 0,Y 355.118,Z 310.252,A -85,B 0,C 180,E1 -13313.181,E2 -13313.181} C_VEL
LIN {X 0,Y 355.245,Z 310.232,A -85,B 0,C 180,E1 -13317.733,E2 -13317.733} C_VEL
LIN {X 0,Y 355.378,Z 310.215,A -85,B 0,C 180,E1 -13320,E2 -13320} C_VEL
LIN {X 0,Y 355.237,Z 310.234,A -85,B 0,C 180,E1 -13322.268,E2 -13322.268} C_VEL
LIN {X 0,Y 355.104,Z 310.254,A -85,B 0,C 180,E1 -13326.82,E2 -13326.82} C_VEL
LIN {X 0,Y 354.96,Z 310.269,A -85,B 0,C 180,E1 -13330.265,E2 -13330.265} C_VEL
LIN {X 0,Y 354.947,Z 310.27,A -85,B 0,C 180,E1 -13334.019,E2 -13334.019} C_VEL
LIN {X 0,Y 354.893,Z 310.277,A -85,B 0,C 180,E1 -13338.092,E2 -13338.092} C_VEL
LIN {X 0,Y 354.819,Z 310.287,A -85,B 0,C 180,E1 -13342.107,E2 -13342.107} C_VEL
LIN {X 0,Y 354.867,Z 310.28,A -85,B 0,C 180,E1 -13345.83,E2 -13345.83} C_VEL
LIN {X 0,Y 354.811,Z 310.287,A -85,B 0,C 180,E1 -13349.683,E2 -13349.683} C_VEL
LIN {X 0,Y 354.834,Z 310.284,A -85,B 0,C 180,E1 -13353.682,E2 -13353.682} C_VEL
LIN {X 0,Y 354.801,Z 310.29,A -85,B 0,C 180,E1 -13356.459,E2 -13356.459} C_VEL
LIN {X 0,Y 354.827,Z 310.285,A -85,B 0,C 180,E1 -13359.424,E2 -13359.424} C_VEL
LIN {X 0,Y 354.791,Z 310.292,A -85,B 0,C 180,E1 -13362.867,E2 -13362.867} C_VEL
LIN {X 0,Y 354.814,Z 310.315,A -85,B 0,C 180,E1 -13365.08,E2 -13365.08} C_VEL
LIN {X 0,Y 355.962,Z 316.642,A -85,B 0,C 180,E1 -13368.613,E2 -13368.613} C_VEL
LIN {X 0,Y 357.118,Z 322.888,A -85,B 0,C 180,E1 -13371.924,E2 -13371.924} C_VEL
LIN {X 0,Y 357.368,Z 326.71,A -85,B 0,C 180,E1 -13373.844,E2 -13373.844} C_VEL
LIN {X 0,Y 356.718,Z 332.316,A -85,B 0,C 180,E1 -13376.519,E2 -13376.519} C_VEL
LIN {X 0,Y 355.775,Z 340.721,A -85,B 0,C 180,E1 -13380.406,E2 -13380.406} C_VEL
LIN {X 0,Y 354.941,Z 349.063,A -85,B 0,C 180,E1 -13384.176,E2 -13384.176} C_VEL
LIN {X 0,Y 354.302,Z 357.375,A -85,B 0,C 180,E1 -13387.859,E2 -13387.859} C_VEL
LIN {X 0,Y 353.998,Z 362.574,A -85,B 0,C 180,E1 -13390.124,E2 -13390.124} C_VEL
LIN {X 0,Y 356.035,Z 377.145,A -85,B 0,C 180,E1 -13390.776,E2 -13390.776} C_VEL
LIN {X 0,Y 357.474,Z 390.27,A -85,B 0,C 180,E1 -13391.59,E2 -13391.59} C_VEL
LIN {X 0,Y 358.306,Z 401.214,A -85,B 0,C 180,E1 -13392.448,E2 -13392.448} C_VEL
LIN {X 0,Y 357.996,Z 407.689,A -85,B 0,C 180,E1 -13393.021,E2 -13393.021} C_VEL
LIN {X 0,Y 356.888,Z 418.393,A -85,B 0,C 180,E1 -13394.143,E2 -13394.143} C_VEL
LIN {X 0,Y 355.876,Z 429.023,A -85,B 0,C 180,E1 -13395.541,E2 -13395.541} C_VEL
LIN {X 0,Y 355.144,Z 437.147,A -85,B 0,C 180,E1 -13396.846,E2 -13396.846} C_VEL
LIN {X 0,Y 354.526,Z 444.556,A -85,B 0,C 180,E1 -13398.276,E2 -13398.276} C_VEL
LIN {X 0,Y 353.937,Z 451.84,A -85,B 0,C 180,E1 -13399.994,E2 -13399.994} C_VEL
LIN {X 0,Y 353.664,Z 456.757,A -85,B 0,C 180,E1 -13401.429,E2 -13401.429} C_VEL
LIN {X 0,Y 353.501,Z 461.517,A -85,B 0,C 180,E1 -13403.149,E2 -13403.149} C_VEL
LIN {X 0,Y 353.433,Z 465.125,A -85,B 0,C 180,E1 -13404.866,E2 -13404.866} C_VEL
LIN {X 0,Y 353.454,Z 467.685,A -85,B 0,C 180,E1 -13406.58,E2 -13406.58} C_VEL
LIN {X 0,Y 353.596,Z 468.874,A -85,B 0,C 180,E1 -13407.722,E2 -13407.722} C_VEL
LIN {X 0,Y 353.6,Z 469.592,A -85,B 0,C 180,E1 -13408.861,E2 -13408.861} C_VEL
LIN {X 0,Y 353.617,Z 469.895,A -85,B 0,C 180,E1 -13410,E2 -13410} C_VEL
LIN {X 0,Y 353.577,Z 469.792,A -85,B 0,C 180,E1 -13411.139,E2 -13411.139} C_VEL
LIN {X 0,Y 353.584,Z 469.29,A -85,B 0,C 180,E1 -13412.278,E2 -13412.278} C_VEL
LIN {X 0,Y 353.426,Z 468.331,A -85,B 0,C 180,E1 -13413.42,E2 -13413.42} C_VEL
LIN {X 0,Y 353.419,Z 466.961,A -85,B 0,C 180,E1 -13414.562,E2 -13414.562} C_VEL
LIN {X 0,Y 353.335,Z 464.662,A -85,B 0,C 180,E1 -13415.997,E2 -13415.997} C_VEL
LIN {X 0,Y 353.542,Z 460.213,A -85,B 0,C 180,E1 -13417.999,E2 -13417.999} C_VEL
LIN {X 0,Y 353.865,Z 455.196,A -85,B 0,C 180,E1 -13419.719,E2 -13419.719} C_VEL
LIN {X 0,Y 354.555,Z 447.769,A -85,B 0,C 180,E1 -13421.723,E2 -13421.723} C_VEL
LIN {X 0,Y 355.472,Z 439.754,A -85,B 0,C 180,E1 -13423.433,E2 -13423.433} C_VEL
LIN {X 0,Y 356.571,Z 430.028,A -85,B 0,C 180,E1 -13425.109,E2 -13425.109} C_VEL
LIN {X 0,Y 357.877,Z 419.685,A -85,B 0,C 180,E1 -13426.544,E2 -13426.544} C_VEL
LIN {X 0,Y 359.289,Z 408.335,A -85,B 0,C 180,E1 -13427.797,E2 -13427.797} C_VEL
LIN {X 0,Y 359.598,Z 400.982,A -85,B 0,C 180,E1 -13428.504,E2 -13428.504} C_VEL
LIN {X 0,Y 359.069,Z 388.916,A -85,B 0,C 180,E1 -13429.51,E2 -13429.51} C_VEL
LIN {X 0,Y 357.698,Z 376.922,A -85,B 0,C 180,E1 -13430.354,E2 -13430.354} C_VEL
LIN {X 0,Y 355.338,Z 364.45,A -85,B 0,C 180,E1 -13431.099,E2 -13431.099} C_VEL
LIN {X 0,Y 354.225,Z 359.211,A -85,B 0,C 180,E1 -13431.376,E2 -13431.376} C_VEL
LIN {X 0,Y 354.811,Z 350.61,A -85,B 0,C 180,E1 -13435.206,E2 -13435.206} C_VEL
LIN {X 0,Y 355.626,Z 342.497,A -85,B 0,C 180,E1 -13438.959,E2 -13438.959} C_VEL
LIN {X 0,Y 356.629,Z 334.569,A -85,B 0,C 180,E1 -13442.816,E2 -13442.816} C_VEL
LIN {X 0,Y 357.563,Z 328.137,A -85,B 0,C 180,E1 -13446.133,E2 -13446.133} C_VEL
LIN {X 0,Y 357.43,Z 324.588,A -85,B 0,C 180,E1 -13448.14,E2 -13448.14} C_VEL
LIN {X 0,Y 356.532,Z 319.254,A -85,B 0,C 180,E1 -13451.491,E2 -13451.491} C_VEL
LIN {X 0,Y 355.657,Z 314.745,A -85,B 0,C 180,E1 -13454.652,E2 -13454.652} C_VEL
LIN {X 0,Y 354.794,Z 310.297,A -85,B 0,C 180,E1 -13458.296,E2 -13458.296} C_VEL
LIN {X 0,Y 354.818,Z 310.294,A -85,B 0,C 180,E1 -13460.666,E2 -13460.666} C_VEL
LIN {X 0,Y 354.825,Z 310.29,A -85,B 0,C 180,E1 -13464.301,E2 -13464.301} C_VEL
LIN {X 0,Y 354.791,Z 310.292,A -85,B 0,C 180,E1 -13467.667,E2 -13467.667} C_VEL
LIN {X 0,Y 354.872,Z 310.282,A -85,B 0,C 180,E1 -13470.621,E2 -13470.621} C_VEL
LIN {X 0,Y 354.904,Z 310.278,A -85,B 0,C 180,E1 -13474.173,E2 -13474.173} C_VEL
LIN {X 0,Y 354.839,Z 310.283,A -85,B 0,C 180,E1 -13477.894,E2 -13477.894} C_VEL
LIN {X 0,Y 354.927,Z 310.273,A -85,B 0,C 180,E1 -13481.891,E2 -13481.891} C_VEL
LIN {X 0,Y 354.947,Z 310.272,A -85,B 0,C 180,E1 -13485.981,E2 -13485.981} C_VEL
LIN {X 0,Y 354.961,Z 310.271,A -85,B 0,C 180,E1 -13489.735,E2 -13489.735} C_VEL
LIN {X 0,Y 355.104,Z 310.251,A -85,B 0,C 180,E1 -13493.18,E2 -13493.18} C_VEL
LIN {X 0,Y 355.248,Z 310.235,A -85,B 0,C 180,E1 -13497.732,E2 -13497.732} C_VEL
LIN {X 0,Y 355.401,Z 310.218,A -85,B 0,C 180,E1 -13500,E2 -13500} C_VEL
LIN {X 0,Y 355.25,Z 310.234,A -85,B 0,C 180,E1 -13502.267,E2 -13502.267} C_VEL
LIN {X 0,Y 355.104,Z 310.254,A -85,B 0,C 180,E1 -13506.82,E2 -13506.82} C_VEL
LIN {X 0,Y 354.896,Z 310.417,A -85,B 0,C 180,E1 -13509.115,E2 -13509.115} C_VEL
LIN {X 0,Y 354.793,Z 312.968,A -85,B 0,C 180,E1 -13512.585,E2 -13512.585} C_VEL
LIN {X 0,Y 354.665,Z 314.768,A -85,B 0,C 180,E1 -13514.928,E2 -13514.928} C_VEL
LIN {X 0,Y 354.584,Z 316.347,A -85,B 0,C 180,E1 -13516.813,E2 -13516.813} C_VEL
LIN {X 0,Y 359.352,Z 329.784,A -85,B 0,C 180,E1 -13517.816,E2 -13517.816} C_VEL
